    upperFelt2StretcherRunFwd   : BOOL;
    upperFelt2StretcherRunRev   : BOOL;

    lowerFeltStretcherRunFwd    : BOOL;
    lowerFeltStretcherRunRev    : BOOL;

    upperInfeedRollRunFwd       : BOOL;
    upperInfeedRollRunRev       : BOOL;

    lowerInfeedRollRunFwd       : BOOL;
    lowerInfeedRollRunRev       : BOOL;

    //────────────────────────────────────────────
    // HMI ALARMS STRUCTURE
    //────────────────────────────────────────────
    hmiAlarms                   : PaperMachine_TypeHmiAlarms; // Alarm structure / Estrutura de alarmes

END_VAR




VAR
 
	instFB_GroupDriveControl_V1 : FB_GroupDriveControl_V1;
	instFB_GroupSpeedControl_V1 : FB_GroupSpeedControl_V1;
	instFB_GroupDisplayFilters_V1 : FB_GroupDisplayFilters_V1;
	instFB_GroupTorqueTrimControl_V1 : FB_GroupTorqueTrimControl_V1;

	instFB_GroupTorqueTrimControl_V2: FB_GroupTorqueTrimControl_V2;
	speedDifError: BOOL;
	speedDifCheck: REAL;
	instTONFeltOverrunDelay: TON;
END_VAR

VAR PERSISTENT

END_VAR

// ─────────────────────────────────────────────────────────────────────────────
// MAIN CALL SEQUENCE
// ─────────────────────────────────────────────────────────────────────────────

_GroupControl();          // 1) State machine: edges, enables, stop modes
_StateDisplay();
_SpeedDifferenceCheck();  // 4) Speed difference monitor & trip
_auxiliaryControls();

_alarmsDisplay();

METHOD _alarmsDisplay
VAR_INPUT
END_VAR
(*
//==============================================================
// FAULT EVALUATION — PER CONDITION (flags only; no global set)
//==============================================================

//----------------------------
// PRESS SECTION DRIVES
//----------------------------
hmiAlarms.pressSectionFirstPressFaultAlarm  := firstPressVfdFaultFeedback;
hmiAlarms.pressSectionSecondPressFaultAlarm := secondPressVfdFaultFeedback;

//----------------------------
// PRESS SECTION AUXILIARIES
//----------------------------
hmiAlarms.pressSectionUpperFeltStretcherFaultAlarm := upperFelt1StretcherFault;
hmiAlarms.pressSectionLowerFeltStretcherFaultAlarm := lowerFeltStretcherFault;
hmiAlarms.pressSectionUpperInfeedRollFaultAlarm    := upperInfeedRollFault;
hmiAlarms.pressSectionLowerInfeedRollFaultAlarm    := lowerInfeedRollFault;


//==============================================================
// PRESS SECTION — FELT EDGE OVERRUN ALARMS (DIRECT SENSORS)
//==============================================================

hmiAlarms.pressSectionUpperFelt1OverrunOperatorSideAlarm := pressSectionUpperFelt1OverrunSensorOperatorSide;
hmiAlarms.pressSectionUpperFelt1OverrunDriveSideAlarm    := pressSectionUpperFelt1OverrunSensorDriveSide;

hmiAlarms.pressSectionUpperFelt2OverrunOperatorSideAlarm := pressSectionUpperFelt2OverrunSensorOperatorSide;
hmiAlarms.pressSectionUpperFelt2OverrunDriveSideAlarm    := pressSectionUpperFelt2OverrunSensorDriveSide;

hmiAlarms.pressSectionLowerFeltOverrunOperatorSideAlarm := pressSectionLowerFeltOverrunSensorOperatorSide;
hmiAlarms.pressSectionLowerFeltOverrunDriveSideAlarm    := pressSectionLowerFeltOverrunSensorDriveSide;


//----------------------------
// PRESS SECTION GROUP FAULT STATUS
//----------------------------
groupFault :=
    hmiAlarms.pressSectionFirstPressFaultAlarm 
	OR hmiAlarms.pressSectionSecondPressFaultAlarm 
	OR hmiAlarms.pressFelt1OverrunOperatorSideAlarm
	OR hmiAlarms.pressFelt1OverrunDriveSideAlarm
	OR hmiAlarms.pressFelt2OverrunOperatorSideAlarm
	OR hmiAlarms.pressFelt2OverrunDriveSideAlarm
	OR hmiAlarms.pressFelt3OverrunOperatorSideAlarm
	OR hmiAlarms.pressFelt3OverrunDriveSideAlarm;


*)
//==============================================================
// FAULT EVALUATION — PER CONDITION (flags only; no global set)
//==============================================================

//----------------------------
// PRESS SECTION DRIVES
//----------------------------
//hmiAlarms.pressSectionFirstPressFaultAlarm  := firstPressVfdFaultFeedback;
//hmiAlarms.pressSectionSecondPressFaultAlarm := secondPressVfdFaultFeedback;

//----------------------------
// PRESS SECTION AUXILIARIES
//----------------------------
hmiAlarms.pressSectionUpperFeltStretcherFaultAlarm := upperFelt1StretcherFault;
hmiAlarms.pressSectionLowerFeltStretcherFaultAlarm := lowerFeltStretcherFault;
hmiAlarms.pressSectionUpperInfeedRollFaultAlarm    := upperInfeedRollFault;
hmiAlarms.pressSectionLowerInfeedRollFaultAlarm    := lowerInfeedRollFault;


//==============================================================
// PRESS SECTION — FELT EDGE OVERRUN ALARMS (DIRECT SENSORS)
//==============================================================

hmiAlarms.pressSectionUpperFelt1OverrunOperatorSideAlarm := pressSectionUpperFelt1OverrunSensorOperatorSide;
hmiAlarms.pressSectionUpperFelt1OverrunDriveSideAlarm    := pressSectionUpperFelt1OverrunSensorDriveSide;

hmiAlarms.pressSectionUpperFelt2OverrunOperatorSideAlarm := pressSectionUpperFelt2OverrunSensorOperatorSide;
hmiAlarms.pressSectionUpperFelt2OverrunDriveSideAlarm    := pressSectionUpperFelt2OverrunSensorDriveSide;

hmiAlarms.pressSectionLowerFeltOverrunOperatorSideAlarm := pressSectionLowerFeltOverrunSensorOperatorSide;
hmiAlarms.pressSectionLowerFeltOverrunDriveSideAlarm    := pressSectionLowerFeltOverrunSensorDriveSide;


//----------------------------
// PRESS SECTION GROUP FAULT STATUS
//----------------------------
groupFault := hmiAlarms.pressSectionFirstPressFaultAlarm OR
		hmiAlarms.pressSectionSecondPressFaultAlarm OR
		hmiAlarms.pressSectionUpperFelt1OverrunOperatorSideAlarm OR
		hmiAlarms.pressSectionUpperFelt1OverrunDriveSideAlarm OR
		hmiAlarms.pressSectionUpperFelt2OverrunOperatorSideAlarm OR
		hmiAlarms.pressSectionUpperFelt2OverrunDriveSideAlarm OR
		hmiAlarms.pressSectionLowerFeltOverrunOperatorSideAlarm OR
		hmiAlarms.pressSectionLowerFeltOverrunDriveSideAlarm;
END_METHOD

METHOD _auxiliaryControls
VAR_INPUT
END_VAR
//============================
// LOWER FELT STRETCHER
//============================
IF NOT lowerFeltStretcherFault THEN
    IF lowerFeltStretcherCmdFwd AND NOT lowerFeltStretcherCmdRev AND NOT lowerFeltStretcherLimitFwd THEN
        lowerFeltStretcherRunFwd := TRUE;
    ELSE
        lowerFeltStretcherRunFwd := FALSE;
    END_IF;

    IF lowerFeltStretcherCmdRev AND NOT lowerFeltStretcherCmdFwd AND NOT lowerFeltStretcherLimitRev THEN
        lowerFeltStretcherRunRev := TRUE;
    ELSE
        lowerFeltStretcherRunRev := FALSE;
    END_IF;
ELSE
    lowerFeltStretcherRunFwd := FALSE;
    lowerFeltStretcherRunRev := FALSE;
END_IF;


//============================
// UPPER INFEED ROLL
//============================
IF NOT upperInfeedRollFault THEN
    IF upperInfeedRollCmdFwd AND NOT upperInfeedRollCmdRev AND NOT upperInfeedRollLimitFwd THEN
        upperInfeedRollRunFwd := TRUE;
    ELSE
        upperInfeedRollRunFwd := FALSE;
    END_IF;

    IF upperInfeedRollCmdRev AND NOT upperInfeedRollCmdFwd AND NOT upperInfeedRollLimitRev THEN
        upperInfeedRollRunRev := TRUE;
    ELSE
        upperInfeedRollRunRev := FALSE;
    END_IF;
ELSE
    upperInfeedRollRunFwd := FALSE;
    upperInfeedRollRunRev := FALSE;
END_IF;


//============================
// LOWER INFEED ROLL
//============================
IF NOT lowerInfeedRollFault THEN
    IF lowerInfeedRollCmdFwd AND NOT lowerInfeedRollCmdRev AND NOT lowerInfeedRollLimitFwd THEN
        lowerInfeedRollRunFwd := TRUE;
    ELSE
        lowerInfeedRollRunFwd := FALSE;
    END_IF;

    IF lowerInfeedRollCmdRev AND NOT lowerInfeedRollCmdFwd AND NOT lowerInfeedRollLimitRev THEN
        lowerInfeedRollRunRev := TRUE;
    ELSE
        lowerInfeedRollRunRev := FALSE;
    END_IF;
ELSE
    lowerInfeedRollRunFwd := FALSE;
    lowerInfeedRollRunRev := FALSE;
END_IF;


//============================
// UPPER FELT 1 STRETCHER
//============================
IF NOT upperFelt1StretcherFault THEN
    IF upperFelt1StretcherCmdFwd AND NOT upperFelt1StretcherCmdRev AND NOT upperFelt1StretcherLimitFwd THEN
        upperFelt1StretcherRunFwd := TRUE;
    ELSE
        upperFelt1StretcherRunFwd := FALSE;
    END_IF;

    IF upperFelt1StretcherCmdRev AND NOT upperFelt1StretcherCmdFwd AND NOT upperFelt1StretcherLimitRev THEN
        upperFelt1StretcherRunRev := TRUE;
    ELSE
        upperFelt1StretcherRunRev := FALSE;
    END_IF;
ELSE
    upperFelt1StretcherRunFwd := FALSE;
    upperFelt1StretcherRunRev := FALSE;
END_IF;

//============================
// UPPER FELT 2 STRETCHER
//============================
IF NOT upperFeltS2tretcherFault THEN
    IF upperFelt2StretcherCmdFwd AND NOT upperFeltt2tretcherCmdRev AND NOT upperFeltS2tretcherLimitFwd THEN
        upperFelt2StretcherRunFwd := TRUE;
    ELSE
        upperFelt2StretcherRunFwd := FALSE;
    END_IF;

    IF upperFeltt2tretcherCmdRev AND NOT upperFelt2StretcherCmdFwd AND NOT upperFeltS2tretcherLimitRev THEN
        upperFelt2StretcherRunRev := TRUE;
    ELSE
        upperFelt2StretcherRunRev := FALSE;
    END_IF;
ELSE
    upperFelt2StretcherRunFwd := FALSE;
    upperFelt2StretcherRunRev := FALSE;
END_IF;
END_METHOD

METHOD _GroupControl
VAR_INPUT
END_VAR
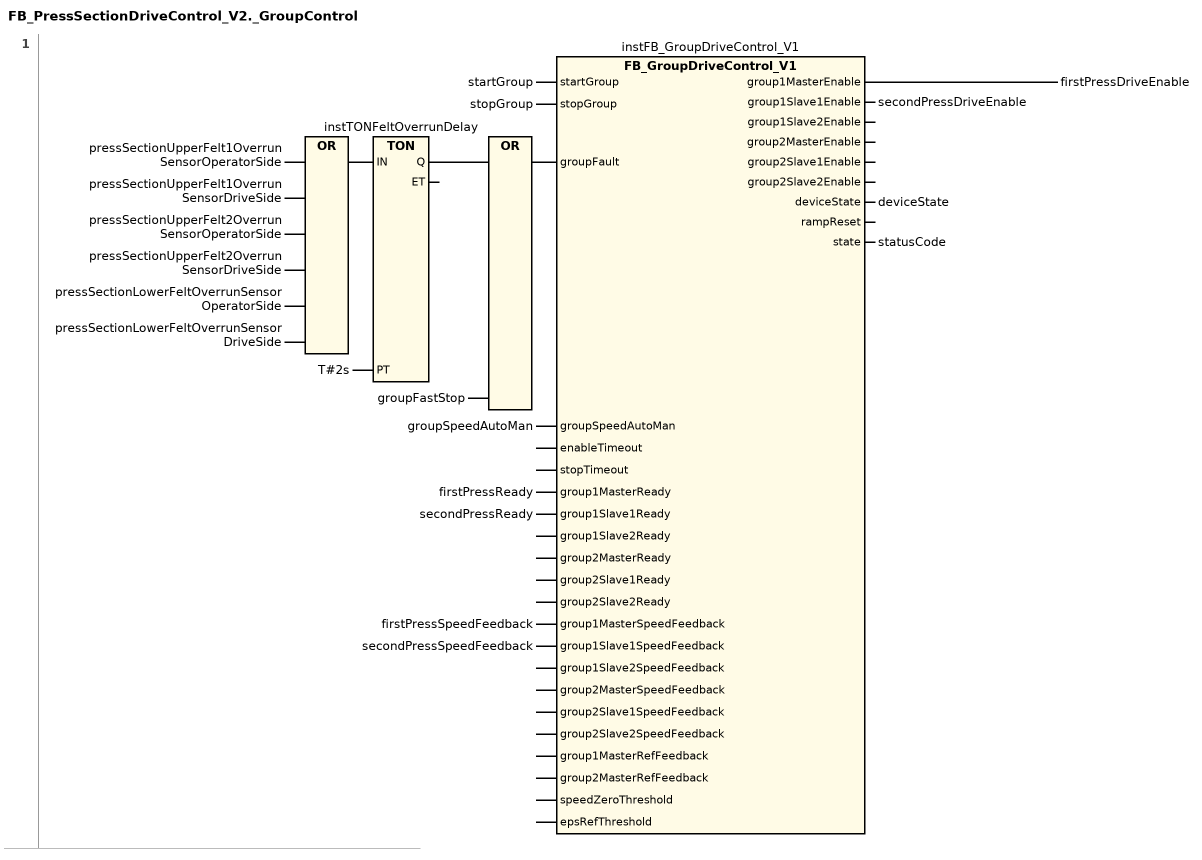
// NETWORK 1
instTONFeltOverrunDelay(IN := pressSectionUpperFelt1OverrunSensorOperatorSide OR pressSectionUpperFelt1OverrunSensorDriveSide OR pressSectionUpperFelt2OverrunSensorOperatorSide OR pressSectionUpperFelt2OverrunSensorDriveSide OR pressSectionLowerFeltOverrunSensorOperatorSide OR pressSectionLowerFeltOverrunSensorDriveSide, PT := T#2s); // TON
instFB_GroupDriveControl_V1(
    startGroup := startGroup,
    stopGroup := stopGroup,
    groupFault := instTONFeltOverrunDelay.Q OR groupFastStop,
    groupSpeedAutoMan := groupSpeedAutoMan,
    group1MasterReady := firstPressReady,
    group1Slave1Ready := secondPressReady,
    group1MasterSpeedFeedback := firstPressSpeedFeedback,
    group1Slave1SpeedFeedback := secondPressSpeedFeedback,
    group1Slave1Enable => secondPressDriveEnable,
    deviceState => deviceState,
    state => statusCode); // FB_GroupDriveControl_V1
firstPressDriveEnable := instFB_GroupDriveControl_V1.group1MasterEnable;

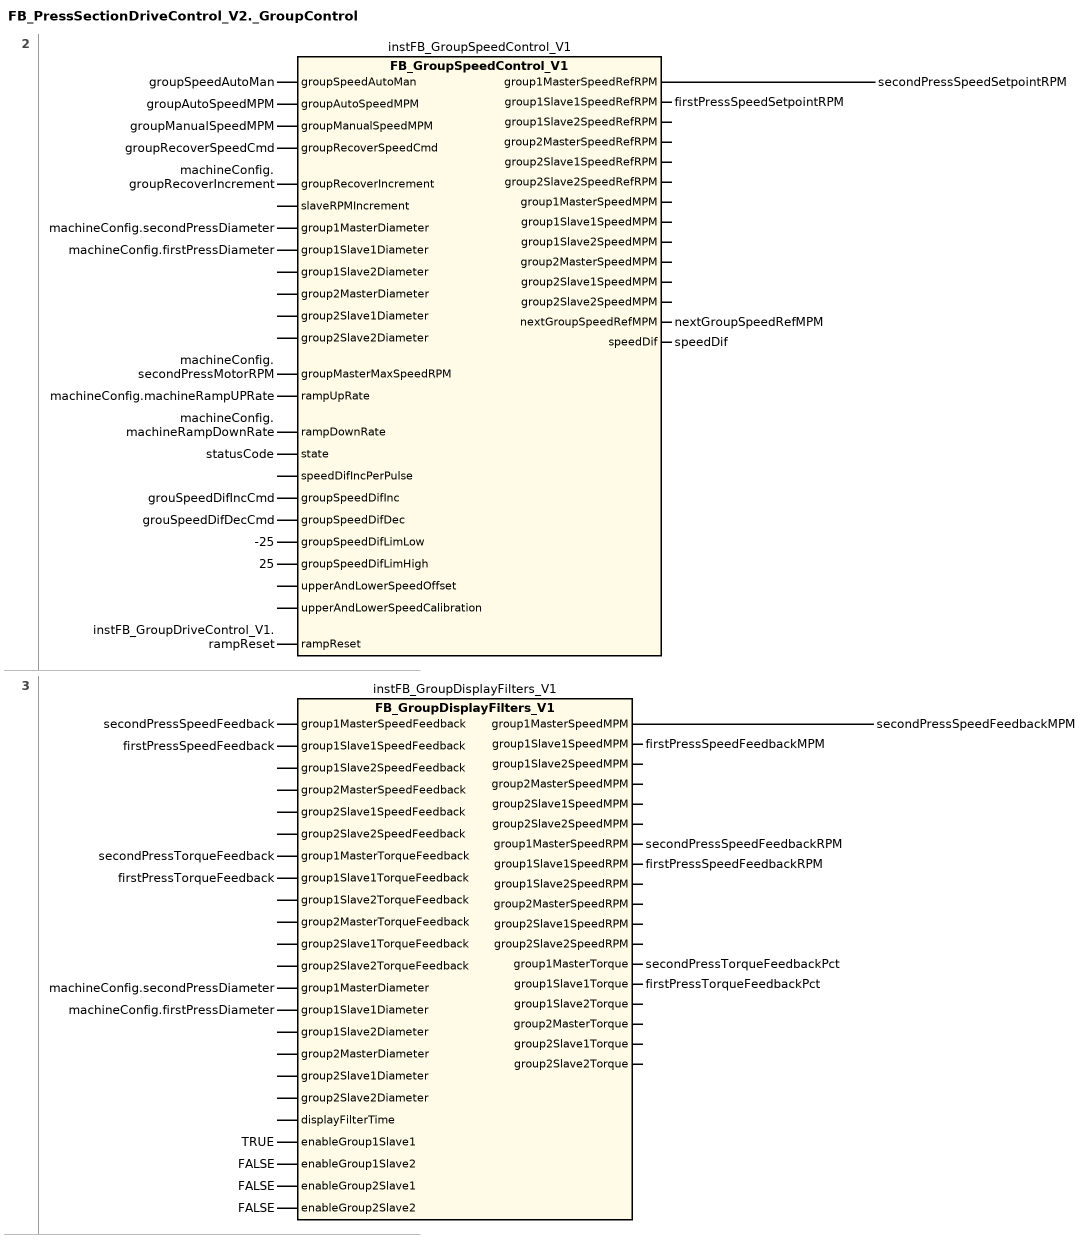
// NETWORK 2
instFB_GroupSpeedControl_V1(
    groupSpeedAutoMan := groupSpeedAutoMan,
    groupAutoSpeedMPM := groupAutoSpeedMPM,
    groupManualSpeedMPM := groupManualSpeedMPM,
    groupRecoverSpeedCmd := groupRecoverSpeedCmd,
    groupRecoverIncrement := machineConfig.groupRecoverIncrement,
    group1MasterDiameter := machineConfig.secondPressDiameter,
    group1Slave1Diameter := machineConfig.firstPressDiameter,
    groupMasterMaxSpeedRPM := machineConfig.secondPressMotorRPM,
    rampUpRate := machineConfig.machineRampUPRate,
    rampDownRate := machineConfig.machineRampDownRate,
    state := statusCode,
    groupSpeedDifInc := grouSpeedDifIncCmd,
    groupSpeedDifDec := grouSpeedDifDecCmd,
    groupSpeedDifLimLow := -25,
    groupSpeedDifLimHigh := 25,
    rampReset := instFB_GroupDriveControl_V1.rampReset,
    group1Slave1SpeedRefRPM => firstPressSpeedSetpointRPM,
    nextGroupSpeedRefMPM => nextGroupSpeedRefMPM,
    speedDif => speedDif); // FB_GroupSpeedControl_V1
secondPressSpeedSetpointRPM := instFB_GroupSpeedControl_V1.group1MasterSpeedRefRPM;

// NETWORK 3
instFB_GroupDisplayFilters_V1(
    group1MasterSpeedFeedback := secondPressSpeedFeedback,
    group1Slave1SpeedFeedback := firstPressSpeedFeedback,
    group1MasterTorqueFeedback := secondPressTorqueFeedback,
    group1Slave1TorqueFeedback := firstPressTorqueFeedback,
    group1MasterDiameter := machineConfig.secondPressDiameter,
    group1Slave1Diameter := machineConfig.firstPressDiameter,
    enableGroup1Slave1 := TRUE,
    enableGroup1Slave2 := FALSE,
    enableGroup2Slave1 := FALSE,
    enableGroup2Slave2 := FALSE,
    group1Slave1SpeedMPM => firstPressSpeedFeedbackMPM,
    group1MasterSpeedRPM => secondPressSpeedFeedbackRPM,
    group1Slave1SpeedRPM => firstPressSpeedFeedbackRPM,
    group1MasterTorque => secondPressTorqueFeedbackPct,
    group1Slave1Torque => firstPressTorqueFeedbackPct); // FB_GroupDisplayFilters_V1
secondPressSpeedFeedbackMPM := instFB_GroupDisplayFilters_V1.group1MasterSpeedMPM;

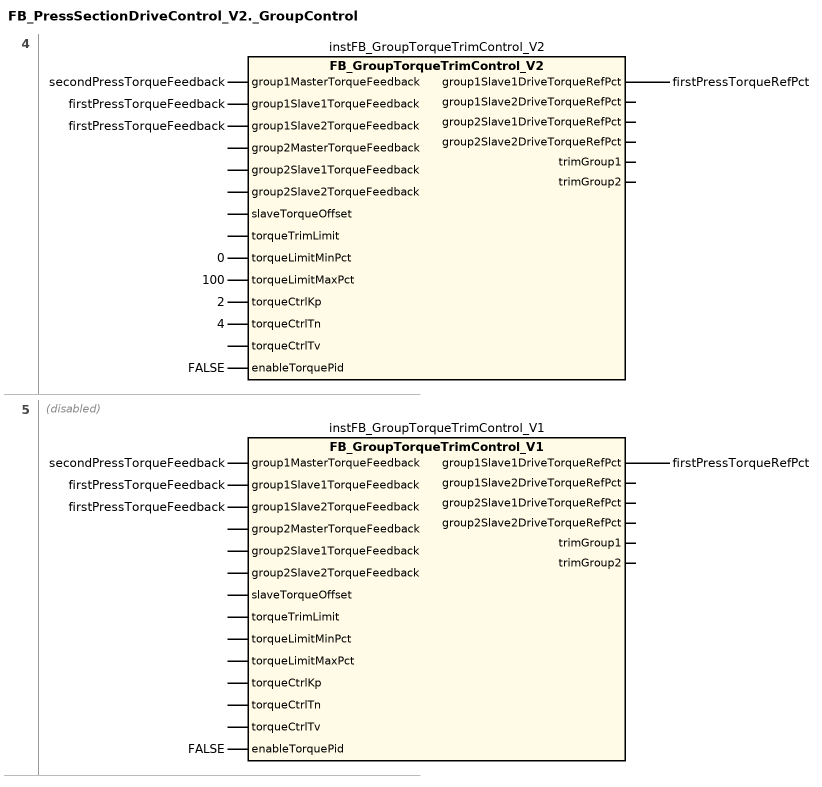
// NETWORK 4
instFB_GroupTorqueTrimControl_V2(
    group1MasterTorqueFeedback := secondPressTorqueFeedback,
    group1Slave1TorqueFeedback := firstPressTorqueFeedback,
    group1Slave2TorqueFeedback := firstPressTorqueFeedback,
    torqueLimitMinPct := 0,
    torqueLimitMaxPct := 100,
    torqueCtrlKp := 2,
    torqueCtrlTn := 4,
    enableTorquePid := FALSE); // FB_GroupTorqueTrimControl_V2
firstPressTorqueRefPct := instFB_GroupTorqueTrimControl_V2.group1Slave1DriveTorqueRefPct;

// NETWORK 5 (disabled)
// instFB_GroupTorqueTrimControl_V1(
//     group1MasterTorqueFeedback := secondPressTorqueFeedback,
//     group1Slave1TorqueFeedback := firstPressTorqueFeedback,
//     group1Slave2TorqueFeedback := firstPressTorqueFeedback,
//     enableTorquePid := FALSE); // FB_GroupTorqueTrimControl_V1
// firstPressTorqueRefPct := instFB_GroupTorqueTrimControl_V1.group1Slave1DriveTorqueRefPct;
END_METHOD

METHOD PRIVATE _Scale : REAL
VAR_INPUT
    X    : REAL;
    I_LO : REAL;
    I_HI : REAL;
    O_LO : REAL;
    O_HI : REAL;
END_VAR
IF I_LO = I_HI THEN
	_Scale := O_LO;
ELSE
	_Scale := (O_HI - O_LO) / (I_HI - I_LO) * (LIMIT(I_LO, X, I_HI) - I_LO) + O_LO;
END_IF;
END_METHOD

// ============================== Methods ==============================
// Intra-section speed supervision for Press Section (firstPress ↔ secondPress)
METHOD _SpeedDifferenceCheck
VAR_INPUT
END_VAR
VAR
    diffPress : REAL;   // Absolute speed difference between master and slave
END_VAR

(*
    //────────────────────────────────────────────
    firstPressSpeedFeedback : REAL; // First press speed feedback / Velocidade medida da prensa 1
    firstPressTorqueFeedback: REAL; // First press torque feedback / Torque da prensa 1
    secondPressSpeedFeedback: REAL; // Second press speed feedback / Velocidade medida da prensa 2
    secondPressTorqueFeedback: REAL; // Second press torque feedback / Torque da prensa 2

*)


speedDifCheck := ABS(secondPressSpeedFeedbackMPM - firstPressSpeedFeedbackMPM);


IF speedDifCheck > 10 THEN
	
	speedDifError := TRUE;
	
	ELSE
		
	speedDifError := FALSE;
	
	
END_IF
END_METHOD

METHOD _StateDisplay
VAR_INPUT
END_VAR

// ──────────────────────────────────────────────────────────────────────────────
// _StateDisplay — Press Section (firstPress = Master, secondPress = Slave)
// Maps the internal machine "state" to a compact HMI status code and derives
// per-drive motor status codes from VFD signals.
//
// statusCode / firstPressStatusCode / secondPressStatusCode legend:
//   0 = Idle, 1 = Starting, 2 = Running, 3 = Fault
//
// Machine "state" groups:
//   0 = IDLE, 1 = ENABLE, 2 = WAIT_EN, 3 = RAMP_EN, 4 = RUN, 5 = STOPPING, 10 = FAULT
// Priority rule (for motors): Fault > Running > Starting > Idle
// ──────────────────────────────────────────────────────────────────────────────
VAR CONSTANT
    STATUS_IDLE     : INT := 0;
    STATUS_STARTING : INT := 1;
    STATUS_RUNNING  : INT := 2;
    STATUS_FAULT    : INT := 3;
END_VAR
(*
// ─────────────── Group machine states into a single HMI statusCode ───────────
CASE state OF
    10: // FAULT
        statusCode := STATUS_FAULT;
    4:  // RUN
        statusCode := STATUS_RUNNING;
    1, 2, 3: // ENABLE / WAIT_EN / RAMP_EN
        statusCode := STATUS_STARTING;
ELSE   // IDLE, STOPPING, or any other
        statusCode := STATUS_IDLE;
END_CASE;


// ─────────────── Per-drive status (priority: Fault > Running > Starting > Idle) ───────────────
// FIRST PRESS (MASTER)
IF firstPressVfdFaultFeedback THEN
    firstPressStatusCode := STATUS_FAULT;
ELSIF firstPressVfdRunFeedback THEN
    firstPressStatusCode := STATUS_RUNNING;
ELSIF firstPressDriveEnable THEN
    firstPressStatusCode := STATUS_STARTING;
ELSE
    firstPressStatusCode := STATUS_IDLE;
END_IF;

// SECOND PRESS (SLAVE)
IF secondPressVfdFaultFeedback THEN
    secondPressStatusCode := STATUS_FAULT;
ELSIF secondPressVfdRunFeedback THEN
    secondPressStatusCode := STATUS_RUNNING;
ELSIF secondPressDriveEnable THEN
    secondPressStatusCode := STATUS_STARTING;
ELSE
    secondPressStatusCode := STATUS_IDLE;
END_IF;
*)
END_METHOD

END_FUNCTION_BLOCK

// ---- Function Blocks/PaperMachine/FB_GroupSpeedControl_V1.TcPOU
FUNCTION_BLOCK FB_GroupSpeedControl_V1
VAR_INPUT
    //==============================================================
    // ─────────────── MODE SELECTION / REFERENCES ───────────────
    //==============================================================
    groupSpeedAutoMan          : BOOL;  // TRUE = Auto, FALSE = Manual
    groupAutoSpeedMPM          : REAL;  // Auto speed reference [m/min]
    groupManualSpeedMPM        : REAL;  // Manual speed reference [m/min]
    groupRecoverSpeedCmd       : BOOL;  // Recover (temporary speed bump)
    groupRecoverIncrement      : REAL;  // Recover increment [m/min]
//    interGroupGearRatio        : REAL;  // Inter-group ratio (next section sync)

	slaveRPMIncrement			: REAL; //Diference in MPM to saturate the speed and enable the torque control

    //==============================================================
    // ─────────────── DIAMETERS (mm) ───────────────
    //==============================================================
    group1MasterDiameter       : REAL;  // Diameter of group 1 master
    group1Slave1Diameter       : REAL;  // Diameter of group 1 slave 1
    group1Slave2Diameter       : REAL;  // Diameter of group 1 slave 2

    group2MasterDiameter       : REAL;  // Diameter of group 2 master
    group2Slave1Diameter       : REAL;  // Diameter of group 2 slave 1
    group2Slave2Diameter       : REAL;  // Diameter of group 2 slave 2

    //==============================================================
    // ─────────────── CONFIGURATION / LIMITS ───────────────
    //==============================================================
    groupMasterMaxSpeedRPM     : REAL;  // Max allowed master RPM
    rampUpRate					: REAL := 0.1;  // Ramp acceleration [RPM/s]
    rampDownRate				: REAL := 0.1;  // Ramp acceleration [RPM/s]
    rampUpRate2					: REAL := 0.1;  // Ramp acceleration [RPM/s]
    rampDownRate2				: REAL := 0.1;  // Ramp acceleration [RPM/s]

	
    state                      : INT;   // Machine state (5 = STOPPING)

	speedDifIncPerPulse		: REAL := 0.05;
	
    groupSpeedDifInc           : BOOL;  // Increment group speed offset
    groupSpeedDifDec           : BOOL;  // Decrement group speed offset
    groupSpeedDifLimLow        : REAL;  // Min offset [%]
    groupSpeedDifLimHigh       : REAL;  // Max offset [%]

    upperAndLowerSpeedOffset   : REAL;  // Bias [%] between group1 and group2
	upperAndLowerSpeedCalibration   : REAL;  // Bias [%] between upper and lower

    rampReset                  : BOOL;  // Reset ramp command
	
	paperPresenceSensor 		: BOOL;
	
END_VAR


VAR_OUTPUT
    //==============================================================
    // ─────────────── FINAL DRIVE SPEEDS (RPM) ───────────────
    //==============================================================
    group1MasterSpeedRefRPM    : REAL;
    group1Slave1SpeedRefRPM    : REAL;
    group1Slave2SpeedRefRPM    : REAL;
    group2MasterSpeedRefRPM    : REAL;
    group2Slave1SpeedRefRPM    : REAL;
    group2Slave2SpeedRefRPM    : REAL;

    //==============================================================
    // ─────────────── SURFACE SPEEDS (MPM) ───────────────
    //==============================================================
    group1MasterSpeedMPM       : REAL;
    group1Slave1SpeedMPM       : REAL;
    group1Slave2SpeedMPM       : REAL;
    group2MasterSpeedMPM       : REAL;
    group2Slave1SpeedMPM       : REAL;
    group2Slave2SpeedMPM       : REAL;

    //==============================================================
    // ─────────────── HANDOFF TO NEXT GROUP ───────────────
    //==============================================================
    nextGroupSpeedRefMPM       : REAL;
	speedDif					: REAL;
	
	
	
END_VAR


VAR
    //==============================================================
    // ─────────────── INTERNAL CALCULATION VARIABLES ───────────────
    //==============================================================
    masterMaxSpeedMPM          : REAL;
    baseCmdSpeedMPM            : REAL;
    cmdSpeedMPM                : REAL;
    targetRPM                  : REAL;
    rampTargetRPM              : REAL;
    baseMasterRefRPM           : REAL;
    groupSpeedOffset           : REAL;
    groupDeltaRatioAll         : REAL;
    upperLowerBiasRatio        : REAL;
    useRamp                    : BOOL;
    epsDiameter                : REAL := 0.001;

    // Gear ratios (set externally or calculated elsewhere)
    group1ToGroup1Slave1Ratio  : REAL := 1.0;
    group1ToGroup1Slave2Ratio  : REAL := 1.0;
    group1ToGroup2MasterRatio  : REAL := 1.0;
    group2ToGroup2Slave1Ratio  : REAL := 1.0;
    group2ToGroup2Slave2Ratio  : REAL := 1.0;

    // Function blocks
    instFB_Gen_SRamp           : FB_Gen_SRamp;
    instFB_SpeedDif_SRamp           : FB_Gen_SRamp;

	rampActive: BOOL;
END_VAR


VAR PERSISTENT
	
    instTUNE2_GroupSpeedDiff   : TUNE2;

END_VAR


(*

IF 	paperPresenceSensor THEN
	//slow	
	instFB_Gen_SRamp.A_UP := MAX(0.0, rampUpRate);
	instFB_Gen_SRamp.A_DN := -MAX(0.0, rampDownRate);

ELSE
	//fast
	instFB_Gen_SRamp.A_UP := MAX(0.0, rampUpRate2);
	instFB_Gen_SRamp.A_DN := -MAX(0.0, rampDownRate2);

END_IF


// Ramp function block execution
instFB_Gen_SRamp(
    X          := rampTargetRPM,
//    A_UP       := MAX(0.0, rampUpRate),
//    A_DN       := -MAX(0.0, rampDownRate),
    VU_MAX     := 1000.0,
    VD_MAX     := -1000.0,
    LIMIT_HIGH := groupMasterMaxSpeedRPM,
    RST        := rampReset);


*)

//==============================================================
// IMPLEMENTATION
//==============================================================

//====================================================================
// ═══ CALL METHOD TO CALCULATE DIAMETER RATIOS ═════════════════════
//====================================================================
_CalculateGearRatios();

//--------------------------------------------------------------
// Calculate master max surface speed [m/min]
//--------------------------------------------------------------
masterMaxSpeedMPM := groupMasterMaxSpeedRPM * (PI * group1MasterDiameter) / 1000.0;


//--------------------------------------------------------------
// Determine base speed source (auto/manual) + Recover bump
//--------------------------------------------------------------
IF groupSpeedAutoMan THEN
    baseCmdSpeedMPM := groupAutoSpeedMPM;
ELSE
    baseCmdSpeedMPM := groupManualSpeedMPM;
END_IF;

IF groupRecoverSpeedCmd THEN
    cmdSpeedMPM := baseCmdSpeedMPM + groupRecoverIncrement;
ELSE
    cmdSpeedMPM := baseCmdSpeedMPM;
END_IF;


//--------------------------------------------------------------
// Convert MPM → target RPM for the master
//--------------------------------------------------------------
targetRPM := _Scale(
    X    := cmdSpeedMPM,
    I_LO := 0.0,
    I_HI := masterMaxSpeedMPM,
    O_LO := 0.0,
    O_HI := groupMasterMaxSpeedRPM);


//--------------------------------------------------------------
// Ramp handling
//--------------------------------------------------------------
IF state = 5 OR state = 0 THEN
    // STOPPING — force ramp down to zero speed
    rampTargetRPM := 0.0;

ELSIF state = 10 THEN
    // FAULT — clear ramp immediately to ensure no residual motion
    rampTargetRPM := 0.0;
//    rampReset     := TRUE;

ELSE
    // Normal operation — ramp follows target speed
    rampTargetRPM := targetRPM;
//    rampReset     := FALSE;
END_IF;

// Detect when a new target speed change requires ramping
IF NOT (rampActive AND ABS(rampTargetRPM - baseMasterRefRPM) >= 1) OR NOT paperPresenceSensor THEN
   rampActive := TRUE; // Rising edge — ramp request detected
 
END_IF;


IF 	paperPresenceSensor THEN
	//slow	
	instFB_Gen_SRamp.A_UP := MAX(0.0, rampUpRate);
	instFB_Gen_SRamp.A_DN := -MAX(0.0, rampDownRate);

ELSE
	//fast
	instFB_Gen_SRamp.A_UP := MAX(0.0, rampUpRate2);
	instFB_Gen_SRamp.A_DN := -MAX(0.0, rampDownRate2);

END_IF


// Ramp function block execution
instFB_Gen_SRamp(
    X          := rampTargetRPM,
//    A_UP       := MAX(0.0, rampUpRate),
//    A_DN       := -MAX(0.0, rampDownRate),
    VU_MAX     := 1000.0,
    VD_MAX     := -1000.0,
    LIMIT_HIGH := groupMasterMaxSpeedRPM,
    RST        := rampReset);


// If ramping, update the baseMasterRefRPM from ramp output
IF rampActive THEN
    baseMasterRefRPM := instFB_Gen_SRamp.Y;

    // Automatically reset ramp flag when the ramp output reaches the target
    IF ABS(instFB_Gen_SRamp.Y - rampTargetRPM) <= 0.05 THEN
        rampActive := FALSE; // Ramp complete
    END_IF;

ELSE
    // No ramping required — direct assignment
    baseMasterRefRPM := rampTargetRPM;
END_IF;


//--------------------------------------------------------------
// Operator offset (TUNE2 control)
//--------------------------------------------------------------
instTUNE2_GroupSpeedDiff(
    SET     := FALSE,
    SU      := groupSpeedDifInc,
    SD      := groupSpeedDifDec,
    RST     := FALSE,
    SS      := speedDifIncPerPulse,
    FS      := speedDifIncPerPulse,
    LIMIT_L := groupSpeedDifLimLow,
    LIMIT_H := groupSpeedDifLimHigh,
    Y       => groupSpeedOffset);


// Ramp function block execution
(*instFB_SpeedDif_SRamp(
    X          := instTUNE2_GroupSpeedDiff.Y,
    A_UP       := MAX(0.0, 0.01),
    A_DN       := -MAX(0.0, 0.01),
    VU_MAX     := 1000.0,
    VD_MAX     := -1000.0,
    LIMIT_HIGH := groupSpeedDifLimHigh,
	LIMIT_LOW := groupSpeedDifLimLow,
    RST        := FALSE,
	Y => groupSpeedOffset);
*)
	
speedDif := groupSpeedOffset;
	
groupDeltaRatioAll  := 1.0 + (groupSpeedOffset * 0.01);
upperLowerBiasRatio := 1.0 + ((upperAndLowerSpeedOffset + upperAndLowerSpeedCalibration) * 0.01);


//--------------------------------------------------------------
// Apply offsets + calculate all drive RPM references
//--------------------------------------------------------------
group1MasterSpeedRefRPM := baseMasterRefRPM * groupDeltaRatioAll;
group1Slave1SpeedRefRPM := group1MasterSpeedRefRPM * group1ToGroup1Slave1Ratio  + slaveRPMIncrement;
group1Slave2SpeedRefRPM := group1MasterSpeedRefRPM * group1ToGroup1Slave2Ratio  + slaveRPMIncrement;

group2MasterSpeedRefRPM := group1MasterSpeedRefRPM * group1ToGroup2MasterRatio * upperLowerBiasRatio;
group2Slave1SpeedRefRPM := group2MasterSpeedRefRPM * group2ToGroup2Slave1Ratio  + slaveRPMIncrement;
group2Slave2SpeedRefRPM := group2MasterSpeedRefRPM * group2ToGroup2Slave2Ratio  + slaveRPMIncrement;


//--------------------------------------------------------------
// Convert RPM → MPM (surface speeds)
//--------------------------------------------------------------
group1MasterSpeedMPM := group1MasterSpeedRefRPM * group1MasterDiameter * PI / 1000.0;
group1Slave1SpeedMPM := (group1Slave1SpeedRefRPM * group1Slave1Diameter * PI / 1000.0);
group1Slave2SpeedMPM := (group1Slave2SpeedRefRPM * group1Slave2Diameter * PI / 1000.0);

group2MasterSpeedMPM := group2MasterSpeedRefRPM * group2MasterDiameter * PI / 1000.0;
group2Slave1SpeedMPM := (group2Slave1SpeedRefRPM * group2Slave1Diameter * PI / 1000.0);
group2Slave2SpeedMPM := (group2Slave2SpeedRefRPM * group2Slave2Diameter * PI / 1000.0);


//--------------------------------------------------------------
// Suggest downstream handoff (group2 master surface speed)
//--------------------------------------------------------------
nextGroupSpeedRefMPM := group1MasterSpeedMPM;


//====================================================================
// ═══ PRIVATE METHOD — CALCULATE DIAMETER RATIOS ════════════════════
//====================================================================
METHOD PRIVATE _CalculateGearRatios
VAR_INPUT
END_VAR

//──────────────────────────────────────────────────────────────
// Gear Ratios — Group 1 (Reference: Group1 Master)
//──────────────────────────────────────────────────────────────
IF group1MasterDiameter > 0.0 THEN
    group1ToGroup2MasterRatio := group1MasterDiameter / group2MasterDiameter;
    group1ToGroup1Slave1Ratio := group1MasterDiameter / group1Slave1Diameter;
    group1ToGroup1Slave2Ratio := group1MasterDiameter / group1Slave2Diameter;
ELSE
    group1ToGroup2MasterRatio := 0.0;
    group1ToGroup1Slave1Ratio := 0.0;
    group1ToGroup1Slave2Ratio := 0.0;
END_IF;

//──────────────────────────────────────────────────────────────
// Gear Ratios — Group 2 (Reference: Group2 Master)
//──────────────────────────────────────────────────────────────
IF group2MasterDiameter > 0.0 THEN
    group2ToGroup2Slave1Ratio := group2MasterDiameter / group2Slave1Diameter;
    group2ToGroup2Slave2Ratio := group2MasterDiameter / group2Slave2Diameter;
ELSE
    group2ToGroup2Slave1Ratio := 0.0;
    group2ToGroup2Slave2Ratio := 0.0;
END_IF;
END_METHOD

METHOD PRIVATE _Scale : REAL
VAR_INPUT
    X    : REAL;
    I_LO : REAL;
    I_HI : REAL;
    O_LO : REAL;
    O_HI : REAL;
END_VAR
IF I_LO = I_HI THEN
	_Scale := O_LO;
ELSE
	_Scale := (O_HI - O_LO) / (I_HI - I_LO) * (LIMIT(I_LO, X, I_HI) - I_LO) + O_LO;
END_IF;
END_METHOD

END_FUNCTION_BLOCK

// ---- Function Blocks/PaperMachine/FB_GroupDisplayFilters_V1.TcPOU
FUNCTION_BLOCK FB_GroupDisplayFilters_V1
VAR_INPUT
    //----------------------------------------------------------------------
    // RAW FEEDBACKS (from drives or sensors)
    //----------------------------------------------------------------------
    group1MasterSpeedFeedback     : REAL;   // [RPM]
    group1Slave1SpeedFeedback     : REAL;   // [RPM]
    group1Slave2SpeedFeedback     : REAL;   // [RPM]
    group2MasterSpeedFeedback     : REAL;   // [RPM]
    group2Slave1SpeedFeedback     : REAL;   // [RPM]
    group2Slave2SpeedFeedback     : REAL;   // [RPM]

    group1MasterTorqueFeedback    : REAL;
    group1Slave1TorqueFeedback    : REAL;
    group1Slave2TorqueFeedback    : REAL;
    group2MasterTorqueFeedback    : REAL;
    group2Slave1TorqueFeedback    : REAL;
    group2Slave2TorqueFeedback    : REAL;

    //----------------------------------------------------------------------
    // DIAMETERS (used to convert RPM → MPM)
    //----------------------------------------------------------------------
    group1MasterDiameter          : REAL;   // [mm]
    group1Slave1Diameter          : REAL;   // [mm]
    group1Slave2Diameter          : REAL;   // [mm]
    group2MasterDiameter          : REAL;   // [mm]
    group2Slave1Diameter          : REAL;   // [mm]
    group2Slave2Diameter          : REAL;   // [mm]

    //----------------------------------------------------------------------
    // FILTER PARAMETERS
    //----------------------------------------------------------------------
    displayFilterTime             : TIME := T#1S;   // EN: Time constant [s]
                                                    // PT: Constante de tempo [s]

    //----------------------------------------------------------------------
    // ENABLE FLAGS (TRUE = filter active)
    //----------------------------------------------------------------------
    enableGroup1Slave1            : BOOL := TRUE;
    enableGroup1Slave2            : BOOL := TRUE;
    enableGroup2Slave1            : BOOL := TRUE;
    enableGroup2Slave2            : BOOL := TRUE;
END_VAR


VAR_OUTPUT
    //----------------------------------------------------------------------
    // SPEEDS IN MPM (converted and filtered)
    //----------------------------------------------------------------------
    group1MasterSpeedMPM : REAL;   // [m/min]
    group1Slave1SpeedMPM : REAL;   // [m/min]
    group1Slave2SpeedMPM : REAL;   // [m/min]
    group2MasterSpeedMPM : REAL;   // [m/min]
    group2Slave1SpeedMPM : REAL;   // [m/min]
    group2Slave2SpeedMPM : REAL;   // [m/min]

    //----------------------------------------------------------------------
    // SPEEDS IN RPM (filtered)
    //----------------------------------------------------------------------
    group1MasterSpeedRPM : REAL;   // [RPM]
    group1Slave1SpeedRPM : REAL;   // [RPM]
    group1Slave2SpeedRPM : REAL;   // [RPM]
    group2MasterSpeedRPM : REAL;   // [RPM]
    group2Slave1SpeedRPM : REAL;   // [RPM]
    group2Slave2SpeedRPM : REAL;   // [RPM]

    //----------------------------------------------------------------------
    // TORQUES (filtered)
    //----------------------------------------------------------------------
    group1MasterTorque : REAL;
    group1Slave1Torque : REAL;
    group1Slave2Torque : REAL;
    group2MasterTorque : REAL;
    group2Slave1Torque : REAL;
    group2Slave2Torque : REAL;
END_VAR


VAR
    //----------------------------------------------------------------------
    // PT1 filter instances
    //----------------------------------------------------------------------
    instPT1_Group1MasterSpeed     : FT_PT1;
    instPT1_Group1Slave1Speed     : FT_PT1;
    instPT1_Group1Slave2Speed     : FT_PT1;
    instPT1_Group2MasterSpeed     : FT_PT1;
    instPT1_Group2Slave1Speed     : FT_PT1;
    instPT1_Group2Slave2Speed     : FT_PT1;

    instPT1_Group1MasterTorque    : FT_PT1;
    instPT1_Group1Slave1Torque    : FT_PT1;
    instPT1_Group1Slave2Torque    : FT_PT1;
    instPT1_Group2MasterTorque    : FT_PT1;
    instPT1_Group2Slave1Torque    : FT_PT1;
    instPT1_Group2Slave2Torque    : FT_PT1;
END_VAR

//────────────────────────────────────────────────────────────
// GROUP 1 — SPEED FILTERS (MPM and RPM)
//────────────────────────────────────────────────────────────
instPT1_Group1MasterSpeed( 
    in := group1MasterSpeedFeedback, 
    T := displayFilterTime, K := 1.0, 
    out => group1MasterSpeedRPM );
group1MasterSpeedMPM := group1MasterSpeedRPM * (group1MasterDiameter * PI / 1000.0);

IF enableGroup1Slave1 THEN
    instPT1_Group1Slave1Speed( in := group1Slave1SpeedFeedback, T := displayFilterTime, K := 1.0, out => group1Slave1SpeedRPM );
ELSE
    group1Slave1SpeedRPM := group1Slave1SpeedFeedback;
END_IF;
group1Slave1SpeedMPM := group1Slave1SpeedRPM * (group1Slave1Diameter * PI / 1000.0);

IF enableGroup1Slave2 THEN
    instPT1_Group1Slave2Speed( in := group1Slave2SpeedFeedback, T := displayFilterTime, K := 1.0, out => group1Slave2SpeedRPM );
ELSE
    group1Slave2SpeedRPM := group1Slave2SpeedFeedback;
END_IF;
group1Slave2SpeedMPM := group1Slave2SpeedRPM * (group1Slave2Diameter * PI / 1000.0);


//────────────────────────────────────────────────────────────
// GROUP 2 — SPEED FILTERS (MPM and RPM)
//────────────────────────────────────────────────────────────
instPT1_Group2MasterSpeed( 
    in := group2MasterSpeedFeedback, 
    T := displayFilterTime, K := 1.0, 
    out => group2MasterSpeedRPM );
group2MasterSpeedMPM := group2MasterSpeedRPM * (group2MasterDiameter * PI / 1000.0);

IF enableGroup2Slave1 THEN
    instPT1_Group2Slave1Speed( in := group2Slave1SpeedFeedback, T := displayFilterTime, K := 1.0, out => group2Slave1SpeedRPM );
ELSE
    group2Slave1SpeedRPM := group2Slave1SpeedFeedback;
END_IF;
group2Slave1SpeedMPM := group2Slave1SpeedRPM * (group2Slave1Diameter * PI / 1000.0);

IF enableGroup2Slave2 THEN
    instPT1_Group2Slave2Speed( in := group2Slave2SpeedFeedback, T := displayFilterTime, K := 1.0, out => group2Slave2SpeedRPM );
ELSE
    group2Slave2SpeedRPM := group2Slave2SpeedFeedback;
END_IF;
group2Slave2SpeedMPM := group2Slave2SpeedRPM * (group2Slave2Diameter * PI / 1000.0);


//────────────────────────────────────────────────────────────
// GROUP 1 — TORQUE FILTERS
//────────────────────────────────────────────────────────────
instPT1_Group1MasterTorque( in := group1MasterTorqueFeedback, T := displayFilterTime, K := 1.0, out => group1MasterTorque );

IF enableGroup1Slave1 THEN
    instPT1_Group1Slave1Torque( in := group1Slave1TorqueFeedback, T := displayFilterTime, K := 1.0, out => group1Slave1Torque );
ELSE
    group1Slave1Torque := group1Slave1TorqueFeedback;
END_IF;

IF enableGroup1Slave2 THEN
    instPT1_Group1Slave2Torque( in := group1Slave2TorqueFeedback, T := displayFilterTime, K := 1.0, out => group1Slave2Torque );
ELSE
    group1Slave2Torque := group1Slave2TorqueFeedback;
END_IF;


//────────────────────────────────────────────────────────────
// GROUP 2 — TORQUE FILTERS
//────────────────────────────────────────────────────────────
instPT1_Group2MasterTorque( in := group2MasterTorqueFeedback, T := displayFilterTime, K := 1.0, out => group2MasterTorque );

IF enableGroup2Slave1 THEN
    instPT1_Group2Slave1Torque( in := group2Slave1TorqueFeedback, T := displayFilterTime, K := 1.0, out => group2Slave1Torque );
ELSE
    group2Slave1Torque := group2Slave1TorqueFeedback;
END_IF;

IF enableGroup2Slave2 THEN
    instPT1_Group2Slave2Torque( in := group2Slave2TorqueFeedback, T := displayFilterTime, K := 1.0, out => group2Slave2Torque );
ELSE
    group2Slave2Torque := group2Slave2TorqueFeedback;
END_IF;

END_FUNCTION_BLOCK

// ---- Function Blocks/PaperMachine/FB_GroupTorqueTrimControl_V1.TcPOU
FUNCTION_BLOCK FB_GroupTorqueTrimControl_V1
VAR_INPUT
    //----------------------------------------------------------------------
    // TORQUE FEEDBACKS (already filtered)
    //----------------------------------------------------------------------
    group1MasterTorqueFeedback     : REAL;  // EN: Master torque feedback [% or Nm]
    group1Slave1TorqueFeedback     : REAL;  // EN: Slave 1 torque feedback [% or Nm]
    group1Slave2TorqueFeedback     : REAL;  // EN: Slave 2 torque feedback [% or Nm]
    group2MasterTorqueFeedback     : REAL;  // EN: Master torque feedback [% or Nm]
    group2Slave1TorqueFeedback     : REAL;  // EN: Slave 1 torque feedback [% or Nm]
    group2Slave2TorqueFeedback     : REAL;  // EN: Slave 2 torque feedback [% or Nm]

    //----------------------------------------------------------------------
    // CONFIGURATION PARAMETERS
    //----------------------------------------------------------------------
    slaveTorqueOffset              : REAL := 0.0;     // EN: Fixed offset between master and slave [%]
    torqueTrimLimit                : REAL := 10.0;    // EN: Max PID trim output [%]
    torqueLimitMinPct              : REAL := -100.0;     // EN: Min torque command limit [%]
    torqueLimitMaxPct              : REAL := 100.0;   // EN: Max torque command limit [%]

    //----------------------------------------------------------------------
    // PID GAINS
    //----------------------------------------------------------------------
    torqueCtrlKp                   : REAL := 1.0;
    torqueCtrlTn                   : REAL := 8.0;
    torqueCtrlTv                   : REAL := 0.0;

    //----------------------------------------------------------------------
    // CONTROL FLAGS
    //----------------------------------------------------------------------
    enableTorquePid                : BOOL := TRUE;    // EN: Enables PID control (FALSE = fixed torque)
END_VAR


VAR_OUTPUT
    //----------------------------------------------------------------------
    // TORQUE REFERENCES (%)
    //----------------------------------------------------------------------
    group1Slave1DriveTorqueRefPct  : REAL;
    group1Slave2DriveTorqueRefPct  : REAL;
    group2Slave1DriveTorqueRefPct  : REAL;
    group2Slave2DriveTorqueRefPct  : REAL;

    //----------------------------------------------------------------------
    // INTERNAL PID OUTPUTS (for monitoring)
    //----------------------------------------------------------------------
    trimGroup1                     : REAL;
    trimGroup2                     : REAL;
	
	
	
END_VAR


VAR
    //----------------------------------------------------------------------
    // INTERNAL PID CONTROLLERS
    //----------------------------------------------------------------------
    instCTRL_PID_Group1TorqueTrim  : CTRL_PID;
    instCTRL_PID_Group2TorqueTrim  : CTRL_PID;

    //----------------------------------------------------------------------
    // INTERNAL SIGNALS
    //----------------------------------------------------------------------
    capMasterGroup1                : REAL;
    capMasterGroup2                : REAL;
    baseLimitGroup1                : REAL;
    baseLimitGroup2                : REAL;
    directTorqueGroup1             : REAL;
    directTorqueGroup2             : REAL;
    avgTorqueGroup1                : REAL;
    avgTorqueGroup2                : REAL;
END_VAR

//======================================================================
// ─── GROUP 1 TORQUE CONTROL ─────────────────────────────────────────
//======================================================================

// Limit master torque safely
capMasterGroup1 := LIMIT(torqueLimitMinPct, group1MasterTorqueFeedback, torqueLimitMaxPct);

// Compute base torque reference for slaves (with offset)
baseLimitGroup1 := group1MasterTorqueFeedback + slaveTorqueOffset;

IF NOT enableTorquePid THEN
    // PID disabled — slaves follow master torque directly
    group1Slave1DriveTorqueRefPct := capMasterGroup1;
    group1Slave2DriveTorqueRefPct := capMasterGroup1;
ELSE
    // PID active — fine trim on torque balance
    directTorqueGroup1 := LIMIT(torqueLimitMinPct, baseLimitGroup1 - torqueTrimLimit, capMasterGroup1);
    avgTorqueGroup1    := 0.5 * (group1Slave1TorqueFeedback + group1Slave2TorqueFeedback);

    instCTRL_PID_Group1TorqueTrim(
        ACT := avgTorqueGroup1,
        SET := baseLimitGroup1,
        MAN := NOT enableTorquePid,
        M_I := 0.0,
        RST := FALSE,
        KP  := torqueCtrlKp,
        TN  := torqueCtrlTn,
        TV  := torqueCtrlTv,
        LL  := torqueLimitMinPct,                   // Bipolar output
        LH  := torqueTrimLimit,
        Y   => trimGroup1
    );

    group1Slave1DriveTorqueRefPct := LIMIT(torqueLimitMinPct, directTorqueGroup1 + trimGroup1, capMasterGroup1);
    group1Slave2DriveTorqueRefPct := LIMIT(torqueLimitMinPct, directTorqueGroup1 + trimGroup1, capMasterGroup1);
END_IF;


//======================================================================
// ─── GROUP 2 TORQUE CONTROL ─────────────────────────────────────────
//======================================================================

capMasterGroup2 := LIMIT(torqueLimitMinPct, group2MasterTorqueFeedback, torqueLimitMaxPct);
baseLimitGroup2 := MIN(
    capMasterGroup2,
    LIMIT(torqueLimitMinPct, group2MasterTorqueFeedback + slaveTorqueOffset, torqueLimitMaxPct)
);

IF NOT enableTorquePid THEN
    group2Slave1DriveTorqueRefPct := capMasterGroup2;
    group2Slave2DriveTorqueRefPct := capMasterGroup2;
ELSE
    directTorqueGroup2 := LIMIT(torqueLimitMinPct, baseLimitGroup2 - torqueTrimLimit, capMasterGroup2);
    avgTorqueGroup2    := 0.5 * (group2Slave1TorqueFeedback + group2Slave2TorqueFeedback);

    instCTRL_PID_Group2TorqueTrim(
        ACT := avgTorqueGroup2,
        SET := baseLimitGroup2,
        MAN := NOT enableTorquePid,
        M_I := 0.0,
        RST := FALSE,
        KP  := torqueCtrlKp,
        TN  := torqueCtrlTn,
        TV  := torqueCtrlTv,
        LL  := 0.0,
        LH  := torqueTrimLimit,
        Y   => trimGroup2
    );

    group2Slave1DriveTorqueRefPct := LIMIT(torqueLimitMinPct, directTorqueGroup2 + trimGroup2, capMasterGroup2);
    group2Slave2DriveTorqueRefPct := LIMIT(torqueLimitMinPct, directTorqueGroup2 + trimGroup2, capMasterGroup2);
END_IF;

END_FUNCTION_BLOCK

// ---- Function Blocks/PaperMachine/FB_GroupTorqueTrimControl_V2.TcPOU
FUNCTION_BLOCK FB_GroupTorqueTrimControl_V2
VAR_INPUT
    //----------------------------------------------------------------------
    // TORQUE FEEDBACKS (already filtered)
    //----------------------------------------------------------------------
    group1MasterTorqueFeedback     : REAL;  // EN: Master torque feedback [% or Nm]
    group1Slave1TorqueFeedback     : REAL;  // EN: Slave 1 torque feedback [% or Nm]
    group1Slave2TorqueFeedback     : REAL;  // EN: Slave 2 torque feedback [% or Nm]
    group2MasterTorqueFeedback     : REAL;  // EN: Master torque feedback [% or Nm]
    group2Slave1TorqueFeedback     : REAL;  // EN: Slave 1 torque feedback [% or Nm]
    group2Slave2TorqueFeedback     : REAL;  // EN: Slave 2 torque feedback [% or Nm]

    //----------------------------------------------------------------------
    // CONFIGURATION PARAMETERS
    //----------------------------------------------------------------------
    slaveTorqueOffset              : REAL := 0.0;     // EN: Fixed offset between master and slave [%]
    torqueTrimLimit                : REAL := 10.0;    // EN: Max PID trim output [%]
    torqueLimitMinPct              : REAL := -10.0;     // EN: Min torque command limit [%]
    torqueLimitMaxPct              : REAL := 10.0;   // EN: Max torque command limit [%]

	
	upperAndLowerDifMinPct :  REAL :=  0.1;
	upperAndLowerDifMaxPct	: REAL := -0.1;
	   
	
    //----------------------------------------------------------------------
    // PID GAINS
    //----------------------------------------------------------------------
    torqueCtrlKp                   : REAL := 1.0;
    torqueCtrlTn                   : REAL := 8.0;
    torqueCtrlTv                   : REAL := 0.0;

    upperAndLowerPIDCtrlKp                   : REAL := 0.10;
    upperAndLowerPIDCtrlTn                   : REAL := 1.0;
    tupperAndLowerPIDCtrlTv                   : REAL := 0.0;
	
	
	enableUpperLowerSpeedTrim			: BOOL;
	
    //----------------------------------------------------------------------
    // CONTROL FLAGS
    //----------------------------------------------------------------------
    enableTorquePid                : BOOL := TRUE;    // EN: Enables PID control (FALSE = fixed torque)
END_VAR


VAR_OUTPUT
    //----------------------------------------------------------------------
    // TORQUE REFERENCES (%)
    //----------------------------------------------------------------------
    group1Slave1DriveTorqueRefPct  : REAL;
    group1Slave2DriveTorqueRefPct  : REAL;
    group2Slave1DriveTorqueRefPct  : REAL;
    group2Slave2DriveTorqueRefPct  : REAL;

    //----------------------------------------------------------------------
    // INTERNAL PID OUTPUTS (for monitoring)
    //----------------------------------------------------------------------
    trimGroup1                     : REAL;
    trimGroup2                     : REAL;
	
	
	upperAndLowerSpeedTrim	 	: REAL;
	
	
END_VAR


VAR
    //----------------------------------------------------------------------
    // INTERNAL PID CONTROLLERS
    //----------------------------------------------------------------------
    instCTRL_PID_Group1TorqueTrim  : CTRL_PID;
    instCTRL_PID_Group2TorqueTrim  : CTRL_PID;
    instCTRL_PID_UpperAndLowerSpdTrim  : CTRL_PID;

	
    //----------------------------------------------------------------------
    // INTERNAL SIGNALS
    //----------------------------------------------------------------------
    capMasterGroup1                : REAL;
    capMasterGroup2                : REAL;
    baseLimitGroup1                : REAL;
    baseLimitGroup2                : REAL;
    directTorqueGroup1             : REAL;
    directTorqueGroup2             : REAL;
    avgTorqueGroup1                : REAL;
    avgTorqueGroup2                : REAL;
	upperAndLowerTorqueDif: REAL;
END_VAR


    instCTRL_PID_Group1TorqueTrim(
        ACT := group1Slave1TorqueFeedback,
        SET := group1MasterTorqueFeedback - slaveTorqueOffset,
        MAN := FALSE,
        M_I := 0.0,
        RST := FALSE,
        KP  := torqueCtrlKp,
        TN  := torqueCtrlTn,
        TV  := torqueCtrlTv,
        LL  := torqueLimitMinPct,                   // Bipolar output
        LH  := torqueLimitMaxPct,
        Y   => group1Slave1DriveTorqueRefPct
    );


	
    instCTRL_PID_Group2TorqueTrim(
        ACT := group2Slave1TorqueFeedback,
        SET := group2MasterTorqueFeedback,
        MAN := FALSE,
        M_I := 0.0,
        RST := FALSE,
        KP  := torqueCtrlKp,
        TN  := torqueCtrlTn,
        TV  := torqueCtrlTv,
        LL  := torqueLimitMinPct,                   // Bipolar output
        LH  := torqueLimitMaxPct,
        Y   => group2Slave1DriveTorqueRefPct
    );


	IF enableUpperLowerSpeedTrim THEN
		
		instCTRL_PID_UpperAndLowerSpdTrim.LL := upperAndLowerDifMinPct;
		instCTRL_PID_UpperAndLowerSpdTrim.LH := upperAndLowerDifMaxPct;
	
	
	ELSE
		
		instCTRL_PID_UpperAndLowerSpdTrim.LL := 0.0;
		instCTRL_PID_UpperAndLowerSpdTrim.LH := 0.0;	
	
	END_IF
	
	
	
		upperAndLowerTorqueDif := group1MasterTorqueFeedback - group2MasterTorqueFeedback;
	
	    instCTRL_PID_UpperAndLowerSpdTrim(
        ACT := upperAndLowerTorqueDif,
        SET := 0,
        MAN := FALSE,
        M_I := 0.0,
        RST := FALSE,
		SUP := 0,
        KP  := upperAndLowerPIDCtrlKp,
        TN  := upperAndLowerPIDCtrlTn,
        TV  := tupperAndLowerPIDCtrlTv,
//        LL  := upperAndLowerDifMinPct,                   // Bipolar output
//        LH  := upperAndLowerDifMaxPct,
        Y   => upperAndLowerSpeedTrim
    );

END_FUNCTION_BLOCK

// ---- Function Blocks/PaperMachine/Auxiliary/FB_SoftstarterWithBypass.TcPOU
FUNCTION_BLOCK FB_SoftstarterWithBypass
VAR_INPUT
    // Commands & interlocks
    startCommand                : BOOL;   // Start command (Comando de partida)
    stopCommand                 : BOOL;   // Stop command (Comando de parada)
    sofstarterOK                : BOOL;   // Softstarter healthy/ready (Softstarter ok/pronto)

    interlock1                  : BOOL;   // External interlock 1 (Intertravamento 1)
    interlock2                  : BOOL;   // External interlock 2 (Intertravamento 2)
    interlock3                  : BOOL;   // External interlock 3 (Intertravamento 3)
    interlock4                  : BOOL;   // External interlock 4 (Intertravamento 4)

    // Feedbacks
    softstarterContactorFb      : BOOL;   // FB - softstarter contactor (Retorno do contator do softstarter)
    lineContactorFb             : BOOL;   // FB - line/bypass contactor (Retorno do contator de linha/bypass)

    // Timers
    startDelayTime              : TIME;   // Ramp-up time before switching to line (Tempo de rampa antes do bypass)
    overlapDelayTime            : TIME;   // Both contactors ON overlap (Sobreposição segura de contatores)
    ssContactorTimeout          : TIME;   // Timeout to get SS contactor FB (Tempo máx. retorno contator softstarter)
    lineContactorTimeout        : TIME;   // Timeout to get Line contactor FB (Tempo máx. retorno contator de linha)

    // Motor current proof
    motorCurrentFeedback        : REAL;   // Measured motor current (Corrente medida do motor)
    minCurrentThreshold         : REAL;   // Minimum current to prove energized (Mínimo para provar energização)
    currentProofTime            : TIME;   // Time current must stay above threshold (Tempo de comprovação)
	
END_VAR

VAR_OUTPUT
	
    faultActive                 : BOOL;   // Latched fault (Falha latched)
    startSequenceRunning        : BOOL;   // Sequence running (Sequência em execução)
    startSequenceFinished       : BOOL;   // Sequence finished successfully (Sequência concluída)

    softstarterContactor        : BOOL;   // CMD softstarter contactor (Comando contator softstarter)
    lineContactor               : BOOL;   // CMD line/bypass contactor (Comando contator linha/bypass)
    softstarterStart            : BOOL;   // CMD start to softstarter (Comando de start do softstarter)

    deviceState                 : STRING(80); // Human-readable state (Estado textual para diagnóstico)
	
END_VAR

VAR
    // State & edges
    step                        : INT;    // State machine step (Etapa)
    startCommandOld             : BOOL;
    rStart                      : BOOL;

    // Timers
    tonStartDelay               : TON;    // Ramp-up timer (Rampa)
    tonOverlapDelay             : TON;    // Overlap timer (Sobreposição)
    tonCurrentProof             : TON;    // Current proof timer (Prova de corrente)

    tonSSFbTimeout              : TON;    // Timeout for SS contactor FB
    tonLineFbTimeout            : TON;    // Timeout for Line contactor FB

    // Helpers
    allInterlocksOK             : BOOL;
	instTONSoftstartDelay: TON;
END_VAR


// ============================ Edges, interlocks, defaults ============================
rStart := startCommand AND NOT startCommandOld;
startCommandOld := startCommand;

allInterlocksOK := interlock1 AND interlock2 AND interlock3 AND interlock4;

// Clear "finished" when a new start is requested or stop asserted
IF rStart OR stopCommand THEN
    startSequenceFinished := FALSE;
END_IF

// Default deviceState (will be overwritten below)
deviceState := 'Idle (Parado)';

// =============================== Fault reset =======================================
// Clear fault when no start request and stop is not held
IF NOT startCommand AND NOT stopCommand THEN
    faultActive := FALSE;
END_IF

// Stop command: immediate safe de-energize (Parada segura imediata)
IF stopCommand THEN
    softstarterStart      := FALSE;
    lineContactor         := FALSE;
    softstarterContactor  := FALSE;

    tonStartDelay(IN:=FALSE);
    tonOverlapDelay(IN:=FALSE);
    tonCurrentProof(IN:=FALSE);
    tonSSFbTimeout(IN:=FALSE);
    tonLineFbTimeout(IN:=FALSE);

    startSequenceRunning  := FALSE;
    step := 0;
END_IF

// ============================= Interlocks & health checks ===========================
// Interlocks must be OK and softstarter OK while sequence
IF startCommand AND NOT allInterlocksOK THEN
    faultActive := TRUE;
    deviceState := 'Fault: interlock open (Falha: intertrav. aberto)';
END_IF

IF startCommand AND NOT sofstarterOK THEN
    faultActive := TRUE;
    deviceState := 'Fault: softstarter not OK (Falha: softstarter NOK)';
END_IF

// If fault is active, do not run sequence
IF faultActive THEN
    softstarterStart      := FALSE;
    lineContactor         := FALSE;
    softstarterContactor  := FALSE;

    tonStartDelay(IN:=FALSE);
    tonOverlapDelay(IN:=FALSE);
    tonCurrentProof(IN:=FALSE);
    tonSSFbTimeout(IN:=FALSE);
    tonLineFbTimeout(IN:=FALSE);

    startSequenceRunning  := FALSE;
    step := 0;
END_IF


// ================================= State machine ===================================
IF startCommand AND NOT faultActive AND sofstarterOK AND allInterlocksOK AND NOT stopCommand THEN
    startSequenceRunning := TRUE;

    CASE step OF
        0: // Idle -> energize softstarter contactor
            deviceState := 'Energizing SS contactor (Acionando contator SS)';
            softstarterContactor := TRUE;

            // timers reset
            tonStartDelay(IN:=FALSE);
            tonOverlapDelay(IN:=FALSE);
            tonCurrentProof(IN:=FALSE);

            // start SS feedback timeout while command is ON and FB is OFF
            tonSSFbTimeout(IN:=NOT softstarterContactorFb, PT:=ssContactorTimeout);

            step := 10;

        10: // Wait SS contactor feedback
            deviceState := 'Waiting SS contactor FB (Aguardando retorno SS)';
            // keep timeout running if still no feedback
            tonSSFbTimeout(IN:=NOT softstarterContactorFb);
			
			instTONSoftstartDelay.PT:=T#5S;
			instTONSoftstartDelay.IN:=TRUE;


            // Timeout fault
            IF tonSSFbTimeout.Q THEN
                faultActive := TRUE;
                deviceState := 'Fault: SS FB timeout (Falha: tempo retorno SS)';
                // force safe
                softstarterStart     := FALSE;
                softstarterContactor := FALSE;
                lineContactor        := FALSE;
                step := 0;
            ELSIF softstarterContactorFb AND instTONSoftstartDelay.Q THEN
                softstarterStart := TRUE;                           // Start softstarter
                tonStartDelay(IN:=TRUE, PT:=startDelayTime);        // Start ramp timer
                tonSSFbTimeout(IN:=FALSE);                          // Stop SS timeout
				instTONSoftstartDelay.IN:=FALSE;

                step := 20;
            END_IF

        20: // Prove motor current while ramping
            deviceState := 'Proving current & ramp (Prova de corrente e rampa)';

            // Current proof: only while current >= threshold
            IF ABS(motorCurrentFeedback) >= minCurrentThreshold THEN
                tonCurrentProof(IN:=TRUE, PT:=currentProofTime);
            ELSE
                tonCurrentProof(IN:=FALSE);
            END_IF

            // Keep ramp timer active
            tonStartDelay(IN:=TRUE);

            // Proceed only when BOTH complete
            IF tonCurrentProof.Q AND tonStartDelay.Q THEN
                deviceState := 'Energizing line contactor (Acionando contator linha)';
                lineContactor := TRUE;

                // start line feedback timeout while command is ON and FB is OFF
                tonLineFbTimeout(IN:=NOT lineContactorFb, PT:=lineContactorTimeout);

                tonCurrentProof(IN:=FALSE); // no longer needed
                step := 30;
            END_IF

        30: // Wait line contactor feedback
            deviceState := 'Waiting line contactor FB (Aguardando retorno linha)';
            // keep timeout running if still no feedback
            tonLineFbTimeout(IN:=NOT lineContactorFb);

            // Timeout fault
            IF tonLineFbTimeout.Q THEN
                faultActive := TRUE;
                deviceState := 'Fault: Line FB timeout (Falha: tempo retorno linha)';
                // safe de-energize SS side and line
                softstarterStart     := FALSE;
                softstarterContactor := FALSE;
                lineContactor        := FALSE;
                step := 0;

            ELSIF lineContactorFb THEN
                deviceState := 'Overlap both contactors (Sobreposição contatores)';
                tonOverlapDelay(IN:=TRUE, PT:=overlapDelayTime); // brief overlap
                tonLineFbTimeout(IN:=FALSE);                     // stop timeout
                step := 40;
            END_IF

        40: // Overlap timing
            deviceState := 'Overlapping... (Sobrepondo...)';
            tonOverlapDelay(IN:=TRUE);
            IF tonOverlapDelay.Q THEN
                softstarterStart     := FALSE;   // Stop softstarter
                softstarterContactor := FALSE;   // Release SS contactor
                tonOverlapDelay(IN:=FALSE);
                deviceState := 'Running on line (Operando em linha)';
                step := 50;
            END_IF

        50: // Running on line
            deviceState := 'Running on line (Operando em linha)';
            startSequenceFinished := TRUE;

            // Stay while start is held; release line on stop
            IF NOT startCommand THEN
                lineContactor := FALSE;
                startSequenceRunning := FALSE;
                deviceState := 'Idle (Parado)';
                step := 0;
            END_IF

        ELSE
            deviceState := 'Idle (Parado)';
            step := 0;
    END_CASE

ELSE
    // No start request / inhibited: ensure safe idle
    startSequenceRunning := FALSE;

    // Keep line latched only if we are in step 50 and startCommand is still ON
    IF step <> 50 THEN
        lineContactor := FALSE;
    END_IF

    // Softstarter side always de-energized when idle
    softstarterStart     := FALSE;
    softstarterContactor := FALSE;

    tonStartDelay(IN:=FALSE);
    tonOverlapDelay(IN:=FALSE);
    tonCurrentProof(IN:=FALSE);
    tonSSFbTimeout(IN:=FALSE);
    tonLineFbTimeout(IN:=FALSE);
	instTONSoftstartDelay(IN:=FALSE);


    IF NOT startCommand THEN
        deviceState := 'Idle (Parado)';
        step := 0;
    END_IF
END_IF

instTONSoftstartDelay();

END_FUNCTION_BLOCK

// ---- Function Blocks/PaperMachine/Auxiliary/FB_MixPumpControl.TcPOU
(*
    FB_MixPumpControl
    - English comments
    - Pressure in mmH2O
    - Uses OSCAT CTRL_PID (v3.33): SUP = DIFF deadband (mmH2O), OFS adds to output Y
    - Includes PV input filter (OSCAT PT1)
    - Includes Jet-to-Wire computation (wire speed in m/min, ratio unitless)
    - Includes ratio tuning via OSCAT TUNE2 (increment/decrement buttons with min/max/step)
    - VFD supervision with RUN feedback timeout
*)

FUNCTION_BLOCK FB_MixPumpControl
VAR_INPUT
    // Commands
    startCommand                : BOOL;          // Start
    stopCommand                 : BOOL;          // Stop

    // Mode
    autoMode                    : BOOL;          // TRUE=Auto / FALSE=Manual

    // Process (pressure in mmH2O)
    pressureFeedback_mmH2O      : REAL;          // Measured pressure [mmH2O]
    manualOutputPct             : REAL;          // Manual output 0..100%

    // Forming board / wire speed and ratio
    formingBoardSpeedMPM        : REAL;          // Wire speed [m/min]
    // Ratio adjust buttons (local HMI)
    jetToWireRatioInc           : BOOL;          // Increment ratio button
    jetToWireRatioDec           : BOOL;          // Decrement ratio button
    // Ratio limits and step
    jetToWireRatioMin           : REAL := 0.50;  // Minimum allowed ratio
    jetToWireRatioMax           : REAL := 2.00;  // Maximum allowed ratio
    jetToWireRatioStep          : REAL := 0.01;  // Step per press

    // Mapping from jet speed to pressure setpoint
    jetHeadGainK                : REAL := 1.0;       // Gain applied to computed head (mmH2O)
    jetHeadOffset_mmH2O         : REAL := 0.0;       // Offset added to computed head (mmH2O)
    minAutoSP_mmH2O             : REAL := 0.0;       // Auto SP clamp low [mmH2O]
    maxAutoSP_mmH2O             : REAL := 4000.0;    // Auto SP clamp high [mmH2O]

    // PID parameters (OSCAT CTRL_PID)
    kp                          : REAL := 0.8;       // Proportional gain
    tn                          : REAL := 3.0;       // Integral time [s]
    tv                          : REAL := 0.0;       // Derivative time [s]
    pidDeadband_mmH2O           : REAL := 5.0;       // SUP: DIFF deadband [mmH2O]

    // Output limits and adjustments (percent)
    outLowLimitPct              : REAL := 0.0;       // Lower output limit [%]
    outHighLimitPct             : REAL := 100.0;     // Upper output limit [%]
    outputOffsetPct             : REAL := 0.0;       // OFS: Output offset [%] added to Y

    // PID housekeeping
    resetPID                    : BOOL;              // Asynchronous reset integrator

    // Input filter (OSCAT PT1) for PV
    enableInputFilter           : BOOL := TRUE;      // TRUE=apply PT1, FALSE=bypass
    inputFilterTime             : TIME := T#300ms;   // PT1 time constant
    inputFilterGainK            : REAL := 1.0;       // PT1 gain (typically 1.0)

    // Interlocks / permissives (4)
    interlock1                  : BOOL;
    interlock2                  : BOOL;
    interlock3                  : BOOL;
    interlock4                  : BOOL;

    // VFD interface & supervision
    vfdReady                    : BOOL;              // VFD ready/healthy
    vfdRunFeedback              : BOOL;              // VFD RUN feedback
    vfdFaultFeedback            : BOOL;              // VFD fault feedback
    vfdRunFbTimeout             : TIME := T#5s;      // Timeout to receive RUN FB after start
END_VAR

VAR_OUTPUT
    // State
    running                     : BOOL;              // TRUE when VFD confirms RUN
    faultActive                 : BOOL;              // Latched fault flag
    deviceState                 : STRING(80);        // Human-readable state
	
    // Commands to VFD
    vfdStartCmd                 : BOOL;              // RUN command
    vfdSpeedPct                 : REAL;              // 0..100% speed reference

    // Telemetry
    jetToWireRatio              : REAL;              // Current ratio value (unitless)
    jetSpeed_mps                : REAL;              // Computed jet speed [m/s]
    headBoxMMH2OCalc          : REAL;              // Auto SP fed to PID [mmH2O]
    headBoxMMH2ORead          : REAL;              // Auto SP fed to PID [mmH2O]
	
    pidDiff                     : REAL;              // CTRL_PID DIFF (deadband-filtered)
    pidLimited                  : BOOL;              // CTRL_PID LIM (Y at limit)
	
	
END_VAR

VAR
    // Edges & helpers
    startOld                    : BOOL;
    rStart                      : BOOL;
    allInterlocksOK             : BOOL;

    // Supervision timer
    tonVfdRunFbTimeout          : TON;

    // Fault text
    faultMsg                    : STRING(80);

    // PID path
    filteredPV_mmH2O            : REAL;
    manualCmdPct                : REAL;
    yPID_Pct                    : REAL;

    // OSCAT instances
    instPID                     : CTRL_PID;         // Pressure controller (percent output)
    instsFT_PT1TInputFilter     : FT_PT1;         // PV PT1 filter
END_VAR


VAR PERSISTENT
	
	instTUNE2RatioSetpoint      : TUNE2;            // Ratio tuner with min/max clamp

END_VAR

// ============================== MAIN EXECUTION ==============================
rStart := startCommand AND NOT startOld;
startOld := startCommand;

allInterlocksOK := interlock1 AND interlock2 AND interlock3 AND interlock4;
deviceState := 'Idle (Stopped)';

// Reset latched fault when idle (no start/stop)
IF NOT startCommand AND NOT stopCommand THEN
    faultActive := FALSE;
    faultMsg := '';
END_IF

// Immediate fault sources
IF vfdFaultFeedback THEN
    faultActive := TRUE;
    faultMsg := 'Fault: VFD fault feedback';
END_IF
IF startCommand AND NOT allInterlocksOK THEN
    faultActive := TRUE;
    faultMsg := 'Fault: interlock open';
END_IF
IF startCommand AND NOT vfdReady THEN
    faultActive := TRUE;
    faultMsg := 'Fault: VFD not ready';
END_IF

// Stop branch (immediate safe stop)
IF stopCommand THEN
    vfdStartCmd := FALSE;
    vfdSpeedPct := 0.0;
    running := FALSE;
    tonVfdRunFbTimeout(IN:=FALSE);
    deviceState := 'Stopping';

ELSE
    // Fault branch (hold safe)
    IF faultActive THEN
        vfdStartCmd := FALSE;
        vfdSpeedPct := 0.0;
        running := FALSE;
        deviceState := faultMsg;
        tonVfdRunFbTimeout(IN:=FALSE);

    // Run branch
    ELSIF startCommand AND allInterlocksOK AND vfdReady THEN
        // --- Ratio tuning via TUNE2 (buttons & min/max clamp) ---
        _RatioInputControl();

        // --- Compute Auto SP (mmH2O) from jet-to-wire and speed ---
        _JetToWire(
            wireSpeedMPM        := formingBoardSpeedMPM,
            ratio               := jetToWireRatio,
            gainK               := jetHeadGainK,
            offset_mmH2O        := jetHeadOffset_mmH2O,
            minSP_mmH2O         := minAutoSP_mmH2O,
            maxSP_mmH2O         := maxAutoSP_mmH2O,
            jetSpeed_mps        => jetSpeed_mps,
            autoSetpoint_mmH2O  => headBoxMMH2OCalc
        );

        // --- Filter PV (mmH2O) with OSCAT PT1 (enable/disable) ---
        _InputFilter(
            enableFilter  := enableInputFilter,
            rawValue      := pressureFeedback_mmH2O,
            filterTime    := inputFilterTime,
            filterGainK   := inputFilterGainK,
            filteredValue => filteredPV_mmH2O
        );

        // --- Manual command in % with clamp ---
        manualCmdPct := manualOutputPct;
        IF manualCmdPct < outLowLimitPct  THEN manualCmdPct := outLowLimitPct;  END_IF;
        IF manualCmdPct > outHighLimitPct THEN manualCmdPct := outHighLimitPct; END_IF;

        // --- OSCAT CTRL_PID (mmH2O domain for ACT/SET, % domain for Y/limits) ---
        instPID(
            ACT := filteredPV_mmH2O,           // PV [mmH2O]
            SET := headBoxMMH2OCalc,         // SP [mmH2O]
            SUP := pidDeadband_mmH2O,          // DIFF deadband [mmH2O]
            OFS := outputOffsetPct,            // Output offset [%]
            M_I := manualCmdPct,               // Manual track value [%]
            MAN := NOT autoMode,               // TRUE => manual (Y = M_I + OFS)
            RST := resetPID,                   // Reset integrator
            KP  := kp,
            TN  := tn,
            TV  := tv,
            LL  := outLowLimitPct,             // Output low limit [%]
            LH  := outHighLimitPct,            // Output high limit [%]
            Y   => yPID_Pct,                   // PID output [%]
            DIFF=> pidDiff,                    // Deadband-filtered DIFF
            LIM => pidLimited                  // TRUE when Y hits limit
        );

        // --- Mode selection & clamp ---
        IF autoMode THEN
            vfdSpeedPct := yPID_Pct;
        ELSE
            vfdSpeedPct := manualCmdPct;
        END_IF
        IF vfdSpeedPct < outLowLimitPct  THEN vfdSpeedPct := outLowLimitPct;  END_IF;
        IF vfdSpeedPct > outHighLimitPct THEN vfdSpeedPct := outHighLimitPct; END_IF;

        // --- Command VFD and supervise RUN FB ---
        vfdStartCmd := TRUE;

        tonVfdRunFbTimeout(
            IN := (vfdStartCmd AND NOT vfdRunFeedback),
            PT := vfdRunFbTimeout
        );

        IF NOT vfdRunFeedback THEN
            deviceState := 'Waiting VFD RUN feedback';
        ELSE
            IF autoMode THEN
                deviceState := 'Running (Auto, pressure in mmH2O)';
            ELSE
                deviceState := 'Running (Manual)';
            END_IF
        END_IF

        IF tonVfdRunFbTimeout.Q THEN
            faultActive := TRUE;
            faultMsg := 'Fault: VFD RUN feedback timeout';
            deviceState := faultMsg;

            vfdStartCmd := FALSE;
            vfdSpeedPct := 0.0;
            running := FALSE;
            tonVfdRunFbTimeout(IN:=FALSE);
        ELSE
            running := vfdRunFeedback;  // running when VFD confirms RUN
        END_IF

    // Idle / safe branch
    ELSE
        vfdStartCmd := FALSE;
        vfdSpeedPct := 0.0;
        running := FALSE;

        IF startCommand AND (NOT allInterlocksOK) THEN
            deviceState := 'Fault: interlock open';
            faultActive := TRUE;
            faultMsg := deviceState;
        ELSIF startCommand AND (NOT vfdReady) THEN
            deviceState := 'Fault: VFD not ready';
            faultActive := TRUE;
            faultMsg := deviceState;
        ELSE
            deviceState := 'Idle (Stopped)';
        END_IF

        tonVfdRunFbTimeout(IN:=FALSE);
    END_IF
END_IF

// ============================================================================
// METHOD: _InputFilter
// OSCAT PT1 filter for PV, with enable/disable and bumpless behavior.
// When disabled, the filter tracks input quickly (tiny T) to avoid bumps.
// ============================================================================
METHOD PRIVATE _InputFilter
VAR_INPUT
    enableFilter   : BOOL;  // TRUE=apply PT1, FALSE=bypass
    rawValue       : REAL;  // Input value to be filtered
    filterTime     : TIME;  // PT1 time constant
    filterGainK    : REAL;  // PT1 gain, typically 1.0
END_VAR
VAR_OUTPUT
    filteredValue  : REAL;  // Filtered (or bypassed) value
END_VAR
VAR
    kUse           : REAL;
    tUse           : TIME;
    yPT1           : REAL;
END_VAR


IF enableFilter THEN
    kUse := filterGainK;
    tUse := filterTime;
ELSE
    // Track input closely for bumpless re-enable
    kUse := 1.0;
    tUse := T#10ms;
END_IF;

instsFT_PT1TInputFilter(
    in  := rawValue,
    T   := tUse,
    K   := kUse,
    out => yPT1
);

// Output selection
IF enableFilter THEN
    filteredValue := yPT1;
ELSE
    filteredValue := rawValue;
END_IF;

//Display filtered value output
headBoxMMH2ORead := yPT1;
END_METHOD

// ============================================================================
// METHOD: _JetToWire
// Computes jet speed from wire speed and ratio, then maps to pressure SP (mmH2O).
// Dynamic head: H[mmH2O] = (v^2 / (2*g)) * 1000, with g = 9.80665 m/s^2.
// A tunable gain/offset is applied; SP is clamped to min/max bounds.
// ============================================================================
METHOD PRIVATE _JetToWire
VAR_INPUT
    wireSpeedMPM        : REAL;  // Wire speed [m/min]
    ratio               : REAL;  // Jet/Wire ratio (unitless), e.g., 1.05
    gainK               : REAL;  // Gain on computed head
    offset_mmH2O        : REAL;  // Offset added to head [mmH2O]
    minSP_mmH2O         : REAL;  // SP lower bound [mmH2O]
    maxSP_mmH2O         : REAL;  // SP upper bound [mmH2O]
END_VAR
VAR_OUTPUT
    jetSpeed_mps        : REAL;  // Jet speed [m/s]
    autoSetpoint_mmH2O  : REAL;  // Pressure SP [mmH2O]
END_VAR
VAR
    wire_mps            : REAL;
    rUse                : REAL;
    dynHead_mmH2O       : REAL;
    cHeadCoeff          : REAL := 50.988; // 1000/(2*g), g=9.80665
END_VAR
// Sanitize ratio
rUse := ratio;
IF rUse < 0.0 THEN rUse := 0.0; END_IF;

// Convert wire speed to m/s
wire_mps := wireSpeedMPM / 60.0;

// Jet speed and dynamic head
jetSpeed_mps := rUse * wire_mps;
dynHead_mmH2O := cHeadCoeff * (jetSpeed_mps * jetSpeed_mps);

// Apply gain/offset and clamp
autoSetpoint_mmH2O := gainK * dynHead_mmH2O + offset_mmH2O;
IF autoSetpoint_mmH2O < minSP_mmH2O THEN autoSetpoint_mmH2O := minSP_mmH2O; END_IF;
IF autoSetpoint_mmH2O > maxSP_mmH2O THEN autoSetpoint_mmH2O := maxSP_mmH2O; END_IF;
END_METHOD

// ============================================================================
// METHOD: _RatioInputControl
// Uses OSCAT TUNE2 to adjust jet-to-wire ratio with buttons, step, min/max.
// The instance preserves ratio value across calls (and download if retained).
// ============================================================================
METHOD PRIVATE _RatioInputControl

instTUNE2RatioSetpoint(
    SET      := FALSE,               // No direct set here (could be mapped to external preset)
    SU       := jetToWireRatioInc,   // Increment button
    SD       := jetToWireRatioDec,   // Decrement button
    RST      := FALSE,               // Optional: add a reset input if needed
    SS       := jetToWireRatioStep,  // Small step per press
    FS       := 0.0,                 // Fast step (unused)
    LIMIT_L  := jetToWireRatioMin,   // Lower bound
    LIMIT_H  := jetToWireRatioMax,   // Upper bound
    Y        => jetToWireRatio       // Current ratio output (unitless)
);
END_METHOD

END_FUNCTION_BLOCK

// ---- Function Blocks/PaperMachine/Auxiliary/FB_FormingBoardRollUpDown.TcPOU
(*---------------------------------------------------------------
  FB_FormingBoardRollUpDown
  Purpose:
    - Drive "Roll Up" / "Roll Down" with safety interlocks
  Behavior:
    - Fault = TRUE  -> both outputs OFF
    - Limit sensors inhibit motion toward that limit
    - If both commands are pressed simultaneously -> no motion
    - Outputs are mutually exclusive
  Notes:
    - Variable names kept exactly as provided (e.g., limitDOwnSensor)
----------------------------------------------------------------*)

FUNCTION_BLOCK FB_FormingBoardRollUpDown
VAR_INPUT
    rollUpCmd      : BOOL;   // Command request to roll UP (active-high)
    rollDownCmd    : BOOL;   // Command request to roll DOWN (active-high)
    limitUpSensor  : BOOL;   // TRUE when upper limit is reached (stop further UP)
    limitDOwnSensor: BOOL;   // TRUE when lower limit is reached (stop further DOWN)
    fault          : BOOL;   // TRUE = fault present -> outputs forced OFF
END_VAR

VAR_OUTPUT
    rollUp         : BOOL;   // Drive UP output (mutually exclusive with rollDown)
    rollDown       : BOOL;   // Drive DOWN output (mutually exclusive with rollUp)
END_VAR

VAR
    // Internal permission and arbitration flags
    upAllowed      : BOOL;
    downAllowed    : BOOL;
    bothPressed    : BOOL;
END_VAR


// 1) Resolve simultaneous commands (prefer safety: do not move)
bothPressed := rollUpCmd AND rollDownCmd;

// 2) Compute permissions considering fault and limit sensors
//    - When a limit sensor is active, inhibit motion further in that direction.
upAllowed   := (NOT fault)
               AND (NOT bothPressed)
               AND rollUpCmd
               AND (NOT limitUpSensor);

downAllowed := (NOT fault)
               AND (NOT bothPressed)
               AND rollDownCmd
               AND (NOT limitDOwnSensor);

// 3) Final outputs (mutually exclusive)
rollUp   := upAllowed  AND (NOT downAllowed);
rollDown := downAllowed AND (NOT upAllowed);

END_FUNCTION_BLOCK

// ---- Function Blocks/PaperMachine/Auxiliary/FB_SimpleMotorStart_V2.TcPOU
FUNCTION_BLOCK FB_SimpleMotorStart_V2
VAR_INPUT
    // ───────── Commands & interlocks ─────────
    startCommand                 : BOOL;   // Pulse to toggle run (Pulso para alternar execução)
    stopCommand                  : BOOL;   // Pulse to force stop (Pulso para forçar parada
	
    motorStarterTrip             : BOOL := TRUE;   // Softstarter healthy/ready (Softstarter ok/pronto)
    safetyOK                   : BOOL	:= TRUE;   // External interlock 1 (Intertravamento 1)
	
    interlock2                   : BOOL := TRUE;   // External interlock 2 (Intertravamento 2)
    interlock3                   : BOOL := TRUE;   // External interlock 3 (Intertravamento 3)
    interlock4                   : BOOL := TRUE;   // External interlock 4 (Intertravamento 4)

    // ───────── Feedbacks ─────────
    softstarterContactorFb       : BOOL := TRUE;   // FB - softstarter contactor
    lineContactorFb              : BOOL := TRUE;   // FB - line/bypass contactor

    // ───────── Timers/thresholds ─────────
    startDelayTime               : TIME;   // Ramp-up time before switching to line
    overlapDelayTime             : TIME;   // Both contactors ON overlap
    ssContactorTimeout           : TIME;   // Timeout to get SS contactor FB
    lineContactorTimeout         : TIME;   // Timeout to get Line contactor FB

    // ───────── Motor current proof ─────────
    motorCurrentFeedback         : REAL;   // Measured motor current
    minCurrentThreshold          : REAL;   // Minimum current to prove energized
    currentProofTime             : TIME;   // Time current must stay above threshold

    // ───────── Pre-start delay for softstarter start ─────────
    softstartStartDelayTime      : TIME;   // Delay before issuing softstarterStart

    // ───────── Motor current filter parameters ─────────
    currentFilterEnable          : BOOL := TRUE;    // Enable current filtering
    currentFilterTime            : TIME := T#200ms; // PT1 time constant
    currentFilterGainK           : REAL := 1.0;     // PT1 gain

    // Optional: choose filtered value for proof logic
    useFilteredForProof          : BOOL := TRUE;    // TRUE uses filtered current for proof
END_VAR

VAR_OUTPUT
    faultActive                  : BOOL;       // Latched fault
    startSequenceRunning         : BOOL;       // Sequence running
    startSequenceFinished        : BOOL;       // Sequence finished successfully

    softstarterContactor         : BOOL;       // CMD softstarter contactor
    lineContactor                : BOOL;       // CMD line/bypass contactor
    softstarterStart             : BOOL;       // CMD start to softstarter

    deviceState                  : STRING(80); // Human-readable state
    statusCode                   : INT;        // 0=Idle, 1=Running, 2=Fault

    motorCurrentFiltered         : REAL;       // Filtered motor current for HMI/logic
END_VAR

VAR
    // ───────── State & edges ─────────
    step                         : INT;    // State machine step
    startCommandOld              : BOOL;
    stopCommandOld               : BOOL;
    rStart                       : BOOL;
    rStop                        : BOOL;

    // ───────── Latch ─────────
    runLatch                     : BOOL;   // Latched run request (start toggles, stop clears)

    // ───────── Timers ─────────
    tonStartDelay                : TON;    // Ramp-up timer
    tonOverlapDelay              : TON;    // Overlap timer
    tonCurrentProof              : TON;    // Current proof timer
    tonSSFbTimeout               : TON;    // Timeout for SS contactor FB
    tonLineFbTimeout             : TON;    // Timeout for Line contactor FB
    instTONSoftstartDelay        : TON;    // Small delay before softstarterStart

    // ───────── Helpers ─────────
    allInterlocksOK              : BOOL;
    proofCurrent                 : REAL;

    // ───────── OSCAT PT1 instance used by _InputFilter ─────────
    // Replace FT_PT1T with the correct type name from your OSCAT lib if different.
    instsFT_PT1TInputFilter      : FT_PT1;

    // Method temp
    _ifFiltered                  : REAL;
END_VAR

// ============================ Edges, interlocks, defaults ============================
rStart := startCommand AND NOT startCommandOld;
rStop  :=  stopCommand AND NOT  stopCommandOld;
startCommandOld := startCommand;
stopCommandOld  := stopCommand;

allInterlocksOK := safetyOK AND interlock2 AND interlock3 AND interlock4;

// Start toggles run latch; Stop forces stop
IF rStart THEN
    runLatch := TRUE;
END_IF;
IF rStop THEN
    runLatch := FALSE;
END_IF;

// Clear "finished" whenever a new start pulse happens or we stop
IF rStart OR rStop THEN
    startSequenceFinished := FALSE;
END_IF;

// Default textual state
deviceState := 'Idle (Parado)';

// =============================== Fault reset =======================================
// Clear fault only when NOT demanding run (latch is OFF) and stop is not held
IF NOT runLatch AND NOT stopCommand THEN
    faultActive := FALSE;
END_IF

// ====================== Filter motor current (for HMI/proof) =======================
THIS^._InputFilter(
    enableFilter := currentFilterEnable,
    rawValue     := motorCurrentFeedback,
    filterTime   := currentFilterTime,
    filterGainK  := currentFilterGainK,
    filteredValue=> _ifFiltered
);
motorCurrentFiltered := _ifFiltered;

proofCurrent := SEL(useFilteredForProof, motorCurrentFeedback, motorCurrentFiltered);

// ============================= Stop handling (immediate) ===========================
IF rStop OR stopCommand THEN
    softstarterStart      := FALSE;
    lineContactor         := FALSE;
    softstarterContactor  := FALSE;

    tonStartDelay(IN:=FALSE);
    tonOverlapDelay(IN:=FALSE);
    tonCurrentProof(IN:=FALSE);
    tonSSFbTimeout(IN:=FALSE);
    tonLineFbTimeout(IN:=FALSE);
    instTONSoftstartDelay(IN:=FALSE);

    startSequenceRunning  := FALSE;
    runLatch := FALSE; // ensure latched run is cleared
    step := 0;
END_IF

// ============================= Interlocks & health checks ===========================
IF runLatch AND NOT allInterlocksOK THEN
    faultActive := TRUE;
    deviceState := 'Fault: interlock open (Falha: intertrav. aberto)';
END_IF

IF runLatch AND NOT motorStarterTrip THEN
    faultActive := TRUE;
    deviceState := 'Fault: softstarter not OK (Falha: softstarter NOK)';
END_IF

// If fault is active, ensure safe idle
IF faultActive THEN
    softstarterStart      := FALSE;
    lineContactor         := FALSE;
    softstarterContactor  := FALSE;

    tonStartDelay(IN:=FALSE);
    tonOverlapDelay(IN:=FALSE);
    tonCurrentProof(IN:=FALSE);
    tonSSFbTimeout(IN:=FALSE);
    tonLineFbTimeout(IN:=FALSE);
    instTONSoftstartDelay(IN:=FALSE);

    startSequenceRunning  := FALSE;
    step := 0;
END_IF

// ================================= State machine ===================================
IF runLatch AND NOT faultActive AND motorStarterTrip AND allInterlocksOK AND NOT stopCommand THEN
    startSequenceRunning := TRUE;

    CASE step OF
        0: // Idle -> energize softstarter contactor
            deviceState := 'Energizing SS contactor (Acionando contator SS)';
            softstarterContactor := TRUE;

            tonStartDelay(IN:=FALSE);
            tonOverlapDelay(IN:=FALSE);
            tonCurrentProof(IN:=FALSE);

            // start SS feedback timeout while command is ON and FB is OFF
            tonSSFbTimeout(IN:=NOT softstarterContactorFb, PT:=ssContactorTimeout);

            step := 10;

        10: // Wait SS contactor feedback, then small delay before SS start
            deviceState := 'Waiting SS FB + pre-start delay (Aguardando retorno SS + atraso)';
            tonSSFbTimeout(IN:=NOT softstarterContactorFb);

            // Pre-start delay parameterized
            IF softstarterContactorFb THEN
                instTONSoftstartDelay(IN:=TRUE, PT:=softstartStartDelayTime);
            ELSE
                instTONSoftstartDelay(IN:=FALSE);
            END_IF

            // Timeout fault
            IF tonSSFbTimeout.Q THEN
                faultActive := TRUE;
                deviceState := 'Fault: SS FB timeout (Falha: tempo retorno SS)';
                softstarterStart     := FALSE;
                softstarterContactor := FALSE;
                lineContactor        := FALSE;
                step := 0;

            ELSIF softstarterContactorFb AND instTONSoftstartDelay.Q THEN
                softstarterStart := TRUE;                           // Start softstarter
                tonStartDelay(IN:=TRUE, PT:=startDelayTime);        // Start ramp timer
                tonSSFbTimeout(IN:=FALSE);                          // Stop SS timeout
                instTONSoftstartDelay(IN:=FALSE);

                step := 20;
            END_IF

        20: // Prove motor current while ramping
            deviceState := 'Proving current & ramp (Prova de corrente e rampa)';

            IF ABS(proofCurrent) >= minCurrentThreshold THEN
                tonCurrentProof(IN:=TRUE, PT:=currentProofTime);
            ELSE
                tonCurrentProof(IN:=FALSE);
            END_IF

            tonStartDelay(IN:=TRUE); // keep ramp timer active

            // Proceed only when BOTH complete
            IF tonCurrentProof.Q AND tonStartDelay.Q THEN
                deviceState := 'Energizing line contactor (Acionando contator linha)';
                lineContactor := TRUE;

                // start line feedback timeout while command is ON and FB is OFF
                tonLineFbTimeout(IN:=NOT lineContactorFb, PT:=lineContactorTimeout);

                tonCurrentProof(IN:=FALSE);
                step := 30;
            END_IF

        30: // Wait line contactor feedback
            deviceState := 'Waiting line contactor FB (Aguardando retorno linha)';
            tonLineFbTimeout(IN:=NOT lineContactorFb);

            IF tonLineFbTimeout.Q THEN
                faultActive := TRUE;
                deviceState := 'Fault: Line FB timeout (Falha: tempo retorno linha)';
                softstarterStart     := FALSE;
                softstarterContactor := FALSE;
                lineContactor        := FALSE;
                step := 0;

            ELSIF lineContactorFb THEN
                deviceState := 'Overlap both contactors (Sobreposição contatores)';
                tonOverlapDelay(IN:=TRUE, PT:=overlapDelayTime);
                tonLineFbTimeout(IN:=FALSE);
                step := 40;
            END_IF

        40: // Overlap timing
            deviceState := 'Overlapping... (Sobrepondo...)';
            tonOverlapDelay(IN:=TRUE);
            IF tonOverlapDelay.Q THEN
                softstarterStart     := FALSE;   // Stop softstarter
                softstarterContactor := FALSE;   // Release SS contactor
                tonOverlapDelay(IN:=FALSE);
                deviceState := 'Running on line (Operando em linha)';
                step := 50;
            END_IF

        50: // Running on line
            deviceState := 'Running on line (Operando em linha)';
            startSequenceFinished := TRUE;

            // Stay running while the latch is set; a new Start pulse toggles it off
            IF NOT runLatch THEN
                lineContactor := FALSE;
                startSequenceRunning := FALSE;
                deviceState := 'Idle (Parado)';
                step := 0;
            END_IF

        ELSE
            deviceState := 'Idle (Parado)';
            step := 0;
    END_CASE

ELSE
    // No latched run / inhibited / fault: ensure safe idle
    startSequenceRunning := FALSE;

    IF step <> 50 THEN
        lineContactor := FALSE;
    END_IF

    softstarterStart     := FALSE;
    softstarterContactor := FALSE;

    tonStartDelay(IN:=FALSE);
    tonOverlapDelay(IN:=FALSE);
    tonCurrentProof(IN:=FALSE);
    tonSSFbTimeout(IN:=FALSE);
    tonLineFbTimeout(IN:=FALSE);
    instTONSoftstartDelay(IN:=FALSE);

    IF NOT runLatch THEN
        deviceState := 'Idle (Parado)';
        step := 0;
    END_IF
END_IF

// =============================== Status code =======================================
IF faultActive THEN
    statusCode := 2;             // Fault
ELSIF startSequenceRunning OR softstarterStart OR lineContactor THEN
    statusCode := 1;             // Running
ELSE
    statusCode := 0;             // Idle
END_IF

// ============================================================================
// METHOD: _InputFilter
// OSCAT PT1 filter for PV, with enable/disable and bumpless behavior.
// When disabled, the filter tracks input quickly (tiny T) to avoid bumps.
// ============================================================================
METHOD PRIVATE _InputFilter
VAR_INPUT
    enableFilter   : BOOL;  // TRUE=apply PT1, FALSE=bypass
    rawValue       : REAL;  // Input value to be filtered
    filterTime     : TIME;  // PT1 time constant
    filterGainK    : REAL;  // PT1 gain, typically 1.0
END_VAR
VAR_OUTPUT
    filteredValue  : REAL;  // Filtered (or bypassed) value
END_VAR
VAR
    kUse           : REAL;
    tUse           : TIME;
    yPT1           : REAL;
END_VAR


IF enableFilter THEN
    kUse := filterGainK;
    tUse := filterTime;
ELSE
    // Track input closely for bumpless re-enable
    kUse := 1.0;
    tUse := T#10ms;
END_IF;

instsFT_PT1TInputFilter(
    in  := rawValue,
    T   := tUse,
    K   := kUse,
    out => yPT1
);

// Output selection
IF enableFilter THEN
    filteredValue := yPT1;
ELSE
    filteredValue := rawValue;
END_IF;
END_METHOD

END_FUNCTION_BLOCK

// ---- Function Blocks/PaperMachine/Auxiliary/FB_SoftstarterWithBypass_V1.TcPOU
FUNCTION_BLOCK FB_SoftstarterWithBypass_V1
VAR_INPUT
    // Commands & interlocks
    startCommand                : BOOL;   // Start pulse (toggle run)
    stopCommand                 : BOOL;   // Stop pulse/level (force stop)
    sofstarterOK                : BOOL;   // Softstarter healthy/ready

    safetyOK                  : BOOL := TRUE;
    interlock2                  : BOOL := TRUE;
    interlock3                  : BOOL := TRUE;
    interlock4                  : BOOL := TRUE;

    // Feedbacks
    softstarterContactorFb      : BOOL;   // FB - softstarter contactor
    lineContactorFb             : BOOL;   // FB - line/bypass contactor

    // Timers
    startDelayTime              : TIME := T#2S;   // Ramp-up time before switching to line
    overlapDelayTime            : TIME := T#3S;   // Both contactors ON overlap
    ssContactorTimeout          : TIME := T#5S;   // Timeout to get SS contactor FB
    lineContactorTimeout        : TIME := T#5S;   // Timeout to get Line contactor FB

    // Motor current proof
    motorCurrentFeedback        : REAL;   // Measured motor current
    minCurrentThreshold         : REAL;   // Minimum current to prove energized
    currentProofTime            : TIME;   // Time current must stay above threshold

    // NEW: Softstarter analog feedback for display
    softstarterCurrentFeedback  : REAL;   // Softstarter phase/line current [A] for HMI
END_VAR

VAR_OUTPUT
    faultActive                 : BOOL;       // Latched fault
    startSequenceRunning        : BOOL;       // Sequence running
    startSequenceFinished       : BOOL;       // Sequence finished successfully

    softstarterContactor        : BOOL;       // CMD softstarter contactor
    lineContactor               : BOOL;       // CMD line/bypass contactor
    softstarterStart            : BOOL;       // CMD start to softstarter

    deviceState                 : STRING(80); // Human-readable state

    // NEW: Status & display values
    statusCode                  : INT;        // 0=Idle, 1=Starting, 2=Running, 3=Fault
    softstarterCurrentDisplay   : REAL;       // Echo of softstarterCurrentFeedback
END_VAR

VAR
    // State & edges
    step                        : INT;    // State machine step
    startCommandOld             : BOOL;
    stopCommandOld              : BOOL;
    rStart                      : BOOL;   // start pulse edge
    rStop                       : BOOL;   // stop pulse edge

    // Run latch toggled by Start pulse
    runLatch                    : BOOL;

    // Timers
    tonStartDelay               : TON;    // Ramp-up timer
    tonOverlapDelay             : TON;    // Overlap timer
    tonCurrentProof             : TON;    // Current proof timer
    tonSSFbTimeout              : TON;    // Timeout for SS contactor FB
    tonLineFbTimeout            : TON;    // Timeout for Line contactor FB
    instTONSoftstartDelay       : TON;    // Small delay before softstarterStart

    // Helpers
    allInterlocksOK             : BOOL;
	
    blinkTon    : TON;   // 1-second timer for blinking / temporizador 1s para piscar
    blinkBit    : BOOL;  // Blink state / estado de pisca	
	
END_VAR

// ============================ Edges, interlocks, defaults ============================
rStart := startCommand AND NOT startCommandOld;
rStop  :=  stopCommand AND NOT  stopCommandOld;
startCommandOld := startCommand;
stopCommandOld  := stopCommand;

allInterlocksOK := safetyOK AND interlock2 AND interlock3 AND interlock4;

// Clear "finished" when a new start request or any stop occurs
IF rStart OR rStop OR stopCommand THEN
    startSequenceFinished := FALSE;
END_IF

// Default state and HMI displays
deviceState := 'Idle (Parado)';
softstarterCurrentDisplay := softstarterCurrentFeedback;

// =============================== Latch / Fault reset =================================
// Start pulse toggles run; Stop pulse/level forces stop and clears latch
IF rStart THEN
    runLatch := TRUE;
END_IF;
IF rStop OR stopCommand THEN
    runLatch := FALSE;
END_IF;

// Clear fault only when not demanding run and stop is not held
IF NOT runLatch AND NOT rStart THEN
    faultActive := FALSE;
END_IF

// ============================= Immediate stop handling ===============================
IF rStop OR stopCommand THEN
    softstarterStart      := FALSE;
    lineContactor         := FALSE;
    softstarterContactor  := FALSE;

    tonStartDelay(IN:=FALSE);
    tonOverlapDelay(IN:=FALSE);
    tonCurrentProof(IN:=FALSE);
    tonSSFbTimeout(IN:=FALSE);
    tonLineFbTimeout(IN:=FALSE);
    instTONSoftstartDelay(IN:=FALSE);

    startSequenceRunning  := FALSE;
    step := 0;
END_IF

// ============================= Interlocks & health checks ============================
IF runLatch AND NOT allInterlocksOK THEN
    faultActive := TRUE;
    deviceState := 'Fault: interlock open (Falha: intertrav. aberto)';
END_IF

IF runLatch AND NOT sofstarterOK THEN
    faultActive := TRUE;
    deviceState := 'Fault: softstarter not OK (Falha: softstarter NOK)';
END_IF

// If fault is active, ensure safe idle
IF faultActive THEN
    softstarterStart      := FALSE;
    lineContactor         := FALSE;
    softstarterContactor  := FALSE;

    tonStartDelay(IN:=FALSE);
    tonOverlapDelay(IN:=FALSE);
    tonCurrentProof(IN:=FALSE);
    tonSSFbTimeout(IN:=FALSE);
    tonLineFbTimeout(IN:=FALSE);
    instTONSoftstartDelay(IN:=FALSE);

    startSequenceRunning  := FALSE;
    step := 0;
END_IF

// ================================= State machine ====================================
IF runLatch AND NOT faultActive AND sofstarterOK AND allInterlocksOK AND NOT stopCommand THEN

    CASE step OF
        0: // Idle -> energize softstarter contactor
		

            deviceState := 'Energizing SS contactor (Acionando contator SS)';
            softstarterContactor := TRUE;

            // reset timers
            tonStartDelay(IN:=FALSE);
            tonOverlapDelay(IN:=FALSE);
            tonCurrentProof(IN:=FALSE);

            // start SS FB timeout while command is ON and FB is OFF
            tonSSFbTimeout(IN:=NOT softstarterContactorFb, PT:=ssContactorTimeout);

            step := 10;

        10: // Wait SS contactor feedback + pre-start delay
		
			startSequenceRunning := TRUE;

            deviceState := 'Waiting SS FB + pre-start delay (Aguardando retorno SS + atraso)';
            tonSSFbTimeout(IN:=NOT softstarterContactorFb);

            // call the small pre-start delay timer every scan
            instTONSoftstartDelay(IN:=softstarterContactorFb, PT:=T#5s);

            // Timeout fault
            IF tonSSFbTimeout.Q THEN
                faultActive := TRUE;
                deviceState := 'Fault: SS FB timeout (Falha: tempo retorno SS)';
                softstarterStart     := FALSE;
                softstarterContactor := FALSE;
                lineContactor        := FALSE;
                step := 0;

            ELSIF softstarterContactorFb AND instTONSoftstartDelay.Q THEN
                softstarterStart := TRUE;                           // Start softstarter
                tonStartDelay(IN:=TRUE, PT:=startDelayTime);        // Start ramp timer
                tonSSFbTimeout(IN:=FALSE);                          // Stop SS timeout
                instTONSoftstartDelay(IN:=FALSE);

                step := 20;
            END_IF

        20: // Prove motor current while ramping
            deviceState := 'Proving current & ramp (Prova de corrente e rampa)';

            IF ABS(motorCurrentFeedback) >= minCurrentThreshold THEN
                tonCurrentProof(IN:=TRUE, PT:=currentProofTime);
            ELSE
                tonCurrentProof(IN:=FALSE);
            END_IF

            tonStartDelay(IN:=TRUE); // keep ramp timer active

            // Proceed only when BOTH complete
            IF tonCurrentProof.Q AND tonStartDelay.Q THEN
                deviceState := 'Energizing line contactor (Acionando contator linha)';
                lineContactor := TRUE;

                // start line feedback timeout while command is ON and FB is OFF
                tonLineFbTimeout(IN:=NOT lineContactorFb, PT:=lineContactorTimeout);

                tonCurrentProof(IN:=FALSE);
                step := 30;
            END_IF

        30: // Wait line contactor feedback
            deviceState := 'Waiting line contactor FB (Aguardando retorno linha)';
            tonLineFbTimeout(IN:=NOT lineContactorFb);

            IF tonLineFbTimeout.Q THEN
                faultActive := TRUE;
                deviceState := 'Fault: Line FB timeout (Falha: tempo retorno linha)';
                softstarterStart     := FALSE;
                softstarterContactor := FALSE;
                lineContactor        := FALSE;
                step := 0;

            ELSIF lineContactorFb THEN
                deviceState := 'Overlap both contactors (Sobreposição contatores)';
                tonOverlapDelay(IN:=TRUE, PT:=overlapDelayTime);
                tonLineFbTimeout(IN:=FALSE);
                step := 40;
            END_IF

        40: // Overlap timing
            deviceState := 'Overlapping... (Sobrepondo...)';
            tonOverlapDelay(IN:=TRUE);
            IF tonOverlapDelay.Q THEN
                softstarterStart     := FALSE;   // Stop softstarter
                softstarterContactor := FALSE;   // Release SS contactor
                tonOverlapDelay(IN:=FALSE);
                deviceState := 'Running on line (Operando em linha)';
                step := 50;
            END_IF

        50: // Running on line
            deviceState := 'Running on line (Operando em linha)';
            startSequenceFinished := TRUE;

            // Stay running while the latch is set; a new Start pulse toggles it off
            IF stopCommand THEN
                lineContactor := FALSE;
                startSequenceRunning := FALSE;
                deviceState := 'Idle (Parado)';
                step := 0;
            END_IF

        ELSE
            deviceState := 'Idle (Parado)';
            step := 0;
    END_CASE

